	            IF "Tor2_RecepturyStacjaMycia".Receptura[#aktualnyNumerReceptury].Krok[#aktualnyKrokMycia].PM[2] = 0
	            THEN
	                ;
	                "Tor2_program".program.numerKroku := 7280;
	                "Tor2_RecepturyStacjaMycia".numerKrokuMycia :=
	                "Tor2_RecepturyStacjaMycia".numerKrokuMycia + 1;
	            END_IF;
	            
	            
	            ;
	            IF "Cip".obiekt["Cip".tor[2].przewodnośćNaPowrocie].WartośćPomiaru <=
	                "Tor2_RecepturyStacjaMycia".Receptura[#aktualnyNumerReceptury].Krok[#aktualnyKrokMycia].PM[12] +
	                "Tor2_RecepturyStacjaMycia".Receptura[#aktualnyNumerReceptury].Krok[#aktualnyKrokMycia].PM[15]
	                
	            THEN
	                "Cip".obiekt["Cip".tor[2].przepływomierzZaWymiennikiem].zerujLicznik1 := 0;
	                "Cip".obiekt["Cip".tor[2].przepływomierzZaWymiennikiem].startLicznik1 := 1;
	            ELSE
	                "Cip".obiekt["Cip".tor[2].przepływomierzZaWymiennikiem].startLicznik1 := 0;
	            END_IF;
	            
	            IF "Cip".obiekt["Cip".tor[2].przepływomierzZaWymiennikiem].licznik1 >
	                "Tor2_RecepturyStacjaMycia".Receptura[#aktualnyNumerReceptury].Krok[#aktualnyKrokMycia].PM[5]
	            THEN
	                "Cip".obiekt["Cip".tor[2].przepływomierzZaWymiennikiem].zerujLicznik1 := 0;
	                "Cip".obiekt["Cip".tor[2].przepływomierzZaWymiennikiem].startLicznik1 := 0;
	              
	                
	                "linia1_pompa_zezwolenie" := 0;
	                "IdźDoKroku"(inNumerKrokuDocelowy := 7271,
	                             inZadaneOpóżnienie := 9,
	                             numerKroku := "Tor2_program".program.numerKroku,
	                             opóźnienie := "Tor2_program".program.opóżnienie,
	                             pauza := "Tor2_hmi".button.bPauza.set);
	                
	                
	              
	            END_IF;
	            
	            
	            "Tor2_program".program.zadana1 := "Tor2_RecepturyStacjaMycia".Receptura[#aktualnyNumerReceptury].Krok[#aktualnyKrokMycia].PM[12] +
	            "Tor2_RecepturyStacjaMycia".Receptura[#aktualnyNumerReceptury].Krok[#aktualnyKrokMycia].PM[15];
	            "Tor2_program".program.aktualna1 := "Cip".obiekt["Cip".tor[2].przewodnośćNaPowrocie].WartośćPomiaru;
	            "Tor2_program".program.zadana2 := "Tor2_RecepturyStacjaMycia".Receptura[#aktualnyNumerReceptury].Krok[#aktualnyKrokMycia].PM[5];
	            "Tor2_program".program.aktualna2 := "Cip".obiekt["Cip".tor[2].przepływomierzZaWymiennikiem].licznik1;
	        7271:
	            
	            "Tor2_RecepturyStacjaMycia".numerKrokuMycia :=
	            "Tor2_RecepturyStacjaMycia".numerKrokuMycia + 1;
	            "Cip".obiekt["Cip".tor[2].przepływomierzZaWymiennikiem].licznik1 := 0;
	            "Tor2_program".program.numerKroku := 7280;
	            
	        7280://Uruchomienie dezynfekcji
	            "Tor2_RecepturyStacjaMycia".numerKrokuMycia := 6;
	            IF "Tor2_RecepturyStacjaMycia".Receptura[#aktualnyNumerReceptury].Krok[#aktualnyKrokMycia].PM[1] = 0
	                OR (#aktualnyKrokMycia = 6 AND "Tor2_hmi".bPomińDesynfekcje)
	            THEN
	                
	                
	                "IdźDoKroku"(inNumerKrokuDocelowy := 7289,
	                             inZadaneOpóżnienie := 30,
	                             numerKroku := "Tor2_program".program.numerKroku,
	                             opóźnienie := "Tor2_program".program.opóżnienie,
	                             pauza := "Tor2_hmi".button.bPauza.set);
	                
	            ELSE
	                "IdźDoKroku"(inNumerKrokuDocelowy := 7281,
	                             inZadaneOpóżnienie := 30,
	                             numerKroku := "Tor2_program".program.numerKroku,
	                             opóźnienie := "Tor2_program".program.opóżnienie,
	                             pauza := "Tor2_hmi".button.bPauza.set);
	            END_IF;
	            
	            
	        7281://napełnianie zbironika dezynfekcji
	            
	            
	            
	            IF "Cip".obiekt["Cip".tor[2].zbiornikDezynfekantu.poziomAnalogowy].WartośćPomiaru > 50
	            THEN
	                
	                
	                "IdźDoKroku"(inNumerKrokuDocelowy := 7282,
	                             inZadaneOpóżnienie := 1,
	                             numerKroku := "Tor2_program".program.numerKroku,
	                             opóźnienie := "Tor2_program".program.opóżnienie,
	                             pauza := "Tor2_hmi".button.bPauza.set);
	            END_IF;
	            "Tor2_program".program.zadana1 := 50;
	            "Tor2_program".program.aktualna1 := "Cip".obiekt["Cip".tor[2].zbiornikDezynfekantu.poziomAnalogowy].WartośćPomiaru;
	            "Tor2_program".program.zadana2 := 0;
	            "Tor2_program".program.aktualna2 := 0;
	            "Cip".obiekt["Cip".tor[2].przepływomierzZaWymiennikiem].licznik1 := 0;
	            
	        7282://dozowanie dezynfekanta
	            "IdźDoKroku"(inNumerKrokuDocelowy := 7283,
	                         inZadaneOpóżnienie := "Tor2_RecepturyStacjaMycia".Receptura[#aktualnyNumerReceptury].Krok[#aktualnyKrokMycia].PM[20],
	                         numerKroku := "Tor2_program".program.numerKroku,
	                         opóźnienie := "Tor2_program".program.opóżnienie,
	                         pauza := "Tor2_hmi".button.bPauza.set);
	            
	            //jeżeli nie leci dezynfekant to kasuj czas dozowania
	            IF "Cip".obiekt["Cip".tor[0].zbiorniczekDozowanieDezynfekantu.czujnikDolnegoPoziomu].hmiPotwWysterowania = 0 THEN
	                "Tor2_program".program.opóżnienie := "Tor2_program".program.opóżnienie - 0.1;
	            END_IF;
	            
	            "Tor2_program".program.zadana1 := "Tor2_RecepturyStacjaMycia".Receptura[#aktualnyNumerReceptury].Krok[#aktualnyKrokMycia].PM[20];
	            "Tor2_program".program.aktualna1 := "Tor2_program".program.opóżnienie;
	            "Tor2_program".program.zadana2 := 0;
	            "Tor2_program".program.aktualna2 := 0;
	            "Cip".obiekt["Cip".tor[2].przepływomierzZaWymiennikiem].licznik1 := 0;
	            
	        7283://dezynfekcja chemiczna
	            "IdźDoKroku"(inNumerKrokuDocelowy := 7284,
	                         inZadaneOpóżnienie := "Tor2_RecepturyStacjaMycia".Receptura[#aktualnyNumerReceptury].Krok[6].PM[6], //czas mycia
	                         numerKroku := "Tor2_program".program.numerKroku,
	                         opóźnienie := "Tor2_program".program.opóżnienie,
	                         pauza := "Tor2_hmi".button.bPauza.set);
	            
	            "Tor2_program".program.zadana1 := "Tor2_RecepturyStacjaMycia".Receptura[#aktualnyNumerReceptury].Krok[6].PM[6];
	            "Tor2_program".program.aktualna1 := "Tor2_program".program.opóżnienie;
	            "Tor2_program".program.zadana2 := 0;
	            "Tor2_program".program.aktualna2 := 0;
	            "Cip".obiekt["Cip".tor[2].przepływomierzZaWymiennikiem].licznik1 := 0;
	            
	        7284://oprożnianie zbiornika dezynfekcji
	            
	            IF "Cip".obiekt["Cip".tor[2].zbiornikDezynfekantu.czujnikDolnegoPoziomu].hmiPotwWysterowania = 0
	            THEN
	                
	                "IdźDoKroku"(inNumerKrokuDocelowy := 7287,
	                             inZadaneOpóżnienie := 2,
	                             numerKroku := "Tor2_program".program.numerKroku,
	                             opóźnienie := "Tor2_program".program.opóżnienie,
	                             pauza := "Tor2_hmi".button.bPauza.set);
	            END_IF;
	            "Tor2_program".program.zadana1 := 0;
	            "Tor2_program".program.aktualna1 := BOOL_TO_INT("Cip".obiekt["Cip".tor[2].zbiornikDezynfekantu.czujnikDolnegoPoziomu].hmiPotwWysterowania);
	            "Tor2_program".program.zadana2 := 0;
	            "Tor2_program".program.aktualna2 := 0;
	            "Cip".obiekt["Cip".tor[2].przepływomierzZaWymiennikiem].licznik1 := 0;
	            
	            
	            
	            
	        7287://Płukanie poo dezynfekcji   
	            
	            
	            IF "Tor2_hmi".bPomińDesynfekcje = 1
	            THEN
	                "Tor2_program".program.numerKroku := 7290;
	            END_IF;
	            
	            "Cip".obiekt["Cip".tor[2].przepływomierzZaWymiennikiem].zerujLicznik1 := 0;
	            "Cip".obiekt["Cip".tor[2].przepływomierzZaWymiennikiem].startLicznik1 := 1;
	            
	            
	            IF "Cip".obiekt["Cip".tor[2].przepływomierzZaWymiennikiem].licznik1 >
	                "Tor2_RecepturyStacjaMycia".Receptura[#aktualnyNumerReceptury].Krok[#aktualnyKrokMycia].PM[5]
	            THEN
	                "Cip".obiekt["Cip".tor[2].przepływomierzZaWymiennikiem].zerujLicznik1 := 0;
	                "Cip".obiekt["Cip".tor[2].przepływomierzZaWymiennikiem].startLicznik1 := 0;
	                "Cip".obiekt["Cip".tor[2].przepływomierzZaWymiennikiem].licznik1 := 0;
	                "Tor2_program".program.numerKroku := 7289;
	            END_IF;
	            
	            
	            
	            "Tor2_program".program.zadana1 := "Tor2_RecepturyStacjaMycia".Receptura[#aktualnyNumerReceptury].Krok[#aktualnyKrokMycia].PM[5];
	            "Tor2_program".program.aktualna1 := "Cip".obiekt["Cip".tor[2].przepływomierzZaWymiennikiem].licznik1;
	            "Tor2_program".program.zadana2 := 0;
	            "Tor2_program".program.aktualna2 := 0;
	            
	        7289://Drenaż zbiornika
	            
	            IF "Tor2_RecepturyStacjaMycia".Receptura[#aktualnyNumerReceptury].Krok[#aktualnyKrokMycia].PM[23] = 0
	            THEN
	                "Tor2_program".program.numerKroku := 7290;
	            END_IF;
	            
	            IF
	                "Cip".obiekt["Cip".tor[2].czujnikPrzepływuNaPowrocie].hmiPotwWysterowania = 1
	            THEN
	                "Tor2_program".program.opóżnienie := 0;
	            END_IF;
	            "IdźDoKroku"(inNumerKrokuDocelowy := 7290,
	                         inZadaneOpóżnienie := "Tor2_RecepturyStacjaMycia".Receptura[#aktualnyNumerReceptury].Krok[#aktualnyKrokMycia].PM[7],
	                         numerKroku := "Tor2_program".program.numerKroku,
	                         opóźnienie := "Tor2_program".program.opóżnienie,
	                         pauza := "Tor2_hmi".button.bPauza.set);
	            
	            "Tor2_program".program.zadana1 := "Tor2_RecepturyStacjaMycia".Receptura[#aktualnyNumerReceptury].Krok[#aktualnyKrokMycia].PM[7];
	            "Tor2_program".program.aktualna1 := "Tor2_program".program.opóżnienie;
	            "Tor2_program".program.zadana2 := 0;
	            "Tor2_program".program.aktualna2 := INT_TO_REAL(BOOL_TO_INT("Cip".obiekt["Cip".tor[2].czujnikPrzepływuNaPowrocie].hmiPotwWysterowania = 1)) * 1.0;
	            
	            
	            
	        7290://zatrzymanie przepływu
	            
	            IF "Cip".obiekt["Cip".tor[2].przepływomierzZaWymiennikiem].WartośćPomiaru <5.0
	            THEN
	                "IdźDoKroku"(inNumerKrokuDocelowy := 7291,
	                             inZadaneOpóżnienie   := 10,
	                             numerKroku           := "Tor2_program".program.numerKroku,
	                             opóźnienie           := "Tor2_program".program.opóżnienie,
	                             pauza:=  "Tor2_hmi".button.bPauza.set);
	            END_IF;
	            
	            "Tor2_program".program.zadana1 := "Tor2_RecepturyStacjaMycia".Receptura[#aktualnyNumerReceptury].Krok[#aktualnyKrokMycia].PM[2];
	            "Tor2_program".program.aktualna1 := "Cip".obiekt["Cip".tor[2].przepływomierzZaWymiennikiem].WartośćPomiaru;
	            "Tor2_program".program.zadana2 :=5;
	            "Tor2_program".program.aktualna2 := "Tor2_program".program.opóżnienie;
	            
	            
	        7291:// odlicz opóźnienie
	            
	            "IdźDoKroku"(inNumerKrokuDocelowy := 7100,
	                         inZadaneOpóżnienie   := 1,
	                         numerKroku           := "Tor2_program".program.numerKroku,
	                         opóźnienie           := "Tor2_program".program.opóżnienie,
	                         pauza:=  "Tor2_hmi".button.bPauza.set);
	            "Tor2_hmi".button.bStop.set := 1;
	          
	            
	            
	        "Tor2_program".program.zadana1 := 0;
	        "Tor2_program".program.aktualna1 :=0;
	        "Tor2_program".program.zadana2 := 10;
	        "Tor2_program".program.aktualna2 := "Tor2_program".program.opóżnienie;
	            
	    7300: //Zaczytanie numeru receptury - krok mycia =2
	        
	        IF "Tor2_RecepturyStacjaMycia".bPokazOknoWyboruReceptury = 0 THEN
	            "Tor2_RecepturyStacjaMycia".bPokazOknoWyboruReceptury := 1;
	        END_IF;
	        IF
	            "Tor2_RecepturyStacjaMycia".klawiszUżyjTejReceptury = 1
	            AND "Tor2_RecepturyStacjaMycia".numerWyswietlanejReceptury = 1
	        THEN
	            "IdźDoKroku"(inNumerKrokuDocelowy := 7301,
	                         inZadaneOpóżnienie   := 0,
	                         numerKroku           := "Tor2_program".program.numerKroku,
	                         opóźnienie           := "Tor2_program".program.opóżnienie,
	                         pauza:=  "Tor2_hmi".button.bPauza.set);
	            "Tor2_RecepturyStacjaMycia".bPokazOknoWyboruReceptury := 0;
	            "Tor2_RecepturyStacjaMycia".numerKrokuMycia := 3;
	            #doSkasowania := 1;
	            
	        END_IF;
	        "Tor2_program".program.zadana1 := 0;
	        "Tor2_program".program.aktualna1 := 0;
	        "Tor2_program".program.zadana2 := 0;
	        "Tor2_program".program.aktualna2 := 0;
	            
	    7301://kolejny krok mycia
	      
	        IF
	            "Tor2_RecepturyStacjaMycia".numerKrokuMycia < 5
	        THEN
	            "IdźDoKroku"(inNumerKrokuDocelowy := 7310,
	                         inZadaneOpóżnienie   := 1,
	                         numerKroku           := "Tor2_program".program.numerKroku,
	                         opóźnienie           := "Tor2_program".program.opóżnienie,
	                         pauza:=  "Tor2_hmi".button.bPauza.set);
	        END_IF;
	        IF
	            "Tor2_RecepturyStacjaMycia".numerKrokuMycia >=5
	        THEN
	            "IdźDoKroku"(inNumerKrokuDocelowy := 7290,
	                         inZadaneOpóżnienie   := 1,
	                         numerKroku           := "Tor2_program".program.numerKroku,
	                         opóźnienie           := "Tor2_program".program.opóżnienie,
	                         pauza:=  "Tor2_hmi".button.bPauza.set);
	            "Tor2_hmi".button.bCip.set := 0;
	        END_IF;
	        "Tor2_program".program.zadana1 := 0;
	        "Tor2_program".program.aktualna1 := 0;
	        "Tor2_program".program.zadana2 := 0;
	        "Tor2_program".program.aktualna2 := 0;
	        
	        
	    7310:// Uzupełnianie poziomu w zbiorniku
	        
	        IF
	            "Tor2_RecepturyStacjaMycia".numerKrokuMycia = 3
	        THEN
	            IF "Cip".obiekt["Cip".tor[0].zbiornikŁugu.czujnikDolnegoPoziomu].hmiPotwWysterowania = 1 THEN
	                "IdźDoKroku"(inNumerKrokuDocelowy := 7320,
	                             inZadaneOpóżnienie   := 1,
	                             numerKroku           := "Tor2_program".program.numerKroku,
	                             opóźnienie           := "Tor2_program".program.opóżnienie,
	                             pauza:=  "Tor2_hmi".button.bPauza.set);
	            END_IF;
	        END_IF;
	        IF
	            "Tor2_RecepturyStacjaMycia".numerKrokuMycia = 4
	        THEN
	            IF "Cip".obiekt["Cip".tor[0].zbiornikKwasu.czujnikDolnegoPoziomu].hmiPotwWysterowania = 1 THEN
	                "IdźDoKroku"(inNumerKrokuDocelowy := 7320,
	                             inZadaneOpóżnienie   := 1,
	                             numerKroku           := "Tor2_program".program.numerKroku,
	                             opóźnienie           := "Tor2_program".program.opóżnienie,
	                             pauza:=  "Tor2_hmi".button.bPauza.set);
	            END_IF;
	        END_IF;
	            
	        "Tor2_program".program.zadana1 :=1;
	        "Tor2_program".program.aktualna1 :=BOOL_TO_INT("Cip".obiekt["Cip".tor[0].zbiornikŁugu.czujnikDolnegoPoziomu].hmiPotwWysterowania);
	        "Tor2_program".program.zadana2 := 1;
	        "Tor2_program".program.aktualna2 := BOOL_TO_INT("Cip".obiekt["Cip".tor[0].zbiornikKwasu.czujnikDolnegoPoziomu].hmiPotwWysterowania);
	        
	    7320://przygotowanie środkla chemicznego
	        
	        IF "Cip".obiekt["Cip".tor[2].przewodnośćNaPowrocie].WartośćPomiaru >=
	            "Tor2_RecepturyStacjaMycia".Receptura[#aktualnyNumerReceptury].Krok[#aktualnyKrokMycia].PM[10] +
	            "Tor2_RecepturyStacjaMycia".Receptura[#aktualnyNumerReceptury].Krok[#aktualnyKrokMycia].PM[15]
	            AND
	            "Cip".obiekt["Cip".tor[2].temperaturaNaPowrocie].WartośćPomiaru >=
	            "Tor2_RecepturyStacjaMycia".Receptura[#aktualnyNumerReceptury].Krok[#aktualnyKrokMycia].PM[13] -
	            "Tor2_RecepturyStacjaMycia".Receptura[#aktualnyNumerReceptury].Krok[#aktualnyKrokMycia].PM[16]
	        THEN
	            "IdźDoKroku"(inNumerKrokuDocelowy := 7321,
	                         inZadaneOpóżnienie   := 30,
	                         numerKroku           := "Tor2_program".program.numerKroku,
	                         opóźnienie           := "Tor2_program".program.opóżnienie,
	                         pauza:=  "Tor2_hmi".button.bPauza.set);
	            
	        END_IF;
	        
	        "Tor2_program".program.zadana1 := "Tor2_RecepturyStacjaMycia".Receptura[#aktualnyNumerReceptury].Krok[#aktualnyKrokMycia].PM[10] +
	        "Tor2_RecepturyStacjaMycia".Receptura[#aktualnyNumerReceptury].Krok[#aktualnyKrokMycia].PM[15];
	        "Tor2_program".program.aktualna1 := "Cip".obiekt["Cip".tor[2].przewodnośćNaPowrocie].WartośćPomiaru;
	        "Tor2_program".program.zadana2 :=  "Tor2_RecepturyStacjaMycia".Receptura[#aktualnyNumerReceptury].Krok[#aktualnyKrokMycia].PM[13] -
	        "Tor2_RecepturyStacjaMycia".Receptura[#aktualnyNumerReceptury].Krok[#aktualnyKrokMycia].PM[16];
	        "Tor2_program".program.aktualna2 := "Cip".obiekt["Cip".tor[2].temperaturaNaPowrocie].WartośćPomiaru;
	        
	        
	        
	    7321://wypłukiwanie środka chemicznego
	        
	        IF "Cip".obiekt["Cip".tor[2].przewodnośćNaPowrocie].WartośćPomiaru <
	            "Tor2_RecepturyStacjaMycia".Receptura[#aktualnyNumerReceptury].Krok[#aktualnyKrokMycia].PM[10] -
	            "Tor2_RecepturyStacjaMycia".Receptura[#aktualnyNumerReceptury].Krok[#aktualnyKrokMycia].PM[15]
	        THEN
	            "IdźDoKroku"(inNumerKrokuDocelowy := 7330,
	                         inZadaneOpóżnienie   := 0,
	                         numerKroku           := "Tor2_program".program.numerKroku,
	                         opóźnienie           := "Tor2_program".program.opóżnienie,
	                         pauza:=  "Tor2_hmi".button.bPauza.set);
	        END_IF;
	        
	        "Tor2_program".program.zadana1 := "Tor2_RecepturyStacjaMycia".Receptura[#aktualnyNumerReceptury].Krok[#aktualnyKrokMycia].PM[10] -
	        "Tor2_RecepturyStacjaMycia".Receptura[#aktualnyNumerReceptury].Krok[#aktualnyKrokMycia].PM[15];
	        "Tor2_program".program.aktualna1 := "Cip".obiekt["Cip".tor[2].przewodnośćNaPowrocie].WartośćPomiaru;
	        "Tor2_program".program.zadana2 := "Tor2_RecepturyStacjaMycia".Receptura[#aktualnyNumerReceptury].Krok[#aktualnyKrokMycia].PM[13] -
	        "Tor2_RecepturyStacjaMycia".Receptura[#aktualnyNumerReceptury].Krok[#aktualnyKrokMycia].PM[16];
	        "Tor2_program".program.aktualna2 := "Cip".obiekt["Cip".tor[2].przewodnośćNaPowrocie].WartośćPomiaru;
	        
	        
	    7330://koniec mycia
	        
	        "IdźDoKroku"(inNumerKrokuDocelowy := 7301,
	                     inZadaneOpóżnienie   := 0,
	                     numerKroku           := "Tor2_program".program.numerKroku,
	                     opóźnienie           := "Tor2_program".program.opóżnienie,
	                     pauza:=  "Tor2_hmi".button.bPauza.set);
	        "Tor2_RecepturyStacjaMycia".numerKrokuMycia :=
	        "Tor2_RecepturyStacjaMycia".numerKrokuMycia + 1;
	        
	        "Tor2_program".program.zadana1 := 0;
	        "Tor2_program".program.aktualna1 := 0;
	        "Tor2_program".program.zadana2 := 0;
	        "Tor2_program".program.aktualna2 := 0;
	        
	    7400://   Zaczytanie numeru receptury (program ustawia Krok mycia = 1) tylko program numer 2
	        
	        IF "Tor2_RecepturyStacjaMycia".bPokazOknoWyboruReceptury = 0 THEN
	            "Tor2_RecepturyStacjaMycia".bPokazOknoWyboruReceptury := 1;
	        END_IF;
	        IF
	            "Tor2_RecepturyStacjaMycia".klawiszUżyjTejReceptury = 1
	            AND "Tor2_RecepturyStacjaMycia".numerWyswietlanejReceptury = 2
	        THEN
	            "IdźDoKroku"(inNumerKrokuDocelowy := 7401,
	                         inZadaneOpóżnienie   := 0,
	                         numerKroku           := "Tor2_program".program.numerKroku,
	                         opóźnienie           := "Tor2_program".program.opóżnienie,
	                         pauza:=  "Tor2_hmi".button.bPauza.set);
	            "Tor2_RecepturyStacjaMycia".bPokazOknoWyboruReceptury := 0;
	            "Tor2_RecepturyStacjaMycia".numerKrokuMycia := 1;
	            #doSkasowania := 1;
	            
	            //Wyskakuje okno wyboru receptur mycia (można wybrać tylko program 2),
	            //po wybraniu krok przechodzi
	            //(program blokuje możliwość pracy na drugim torze - może mrygać na nim kontrolka CIP)
	            //do zrobienia !!!!!
	            
	            
	        END_IF;
	        "Tor2_program".program.zadana1 := 0;
	        "Tor2_program".program.aktualna1 := 0;
	        "Tor2_program".program.zadana2 := 0;
	        "Tor2_program".program.aktualna2 := 0;
	        
	        
	    7401:// drenaż zbiornika wody wtórnej
	        
	        
	        IF
	            "Cip".obiekt["Cip".tor[2].czujnikPrzepływuNaPowrocie].hmiPotwWysterowania = 1
	        THEN
	            "Tor2_program".program.opóżnienie := 0;
	        END_IF;
	        "IdźDoKroku"(inNumerKrokuDocelowy := 7402,
	                     inZadaneOpóżnienie   := "Tor2_RecepturyStacjaMycia".Receptura[#aktualnyNumerReceptury].Krok[#aktualnyKrokMycia].PM[7],
	                     numerKroku           := "Tor2_program".program.numerKroku,
	                     opóźnienie           := "Tor2_program".program.opóżnienie,
	                     pauza:=  "Tor2_hmi".button.bPauza.set);
	        
	        "Tor2_program".program.zadana1 := "Tor2_RecepturyStacjaMycia".Receptura[#aktualnyNumerReceptury].Krok[#aktualnyKrokMycia].PM[7];
	        "Tor2_program".program.aktualna1 := "Tor2_program".program.opóżnienie;
	        "Tor2_program".program.zadana2 := 0;
	        "Tor2_program".program.aktualna2 := INT_TO_REAL(BOOL_TO_INT("Cip".obiekt["Cip".tor[2].czujnikPrzepływuNaPowrocie].hmiPotwWysterowania = 1)) * 1.0;
	        
	    7402://płukanie zimne
	            
	        IF "Tor2_RecepturyStacjaMycia".Receptura[#aktualnyNumerReceptury].Krok[#aktualnyKrokMycia].PM[2] = 0
	            THEN
	                ;
	                "Tor2_program".program.numerKroku := 7403;
	                "Tor2_RecepturyStacjaMycia".numerKrokuMycia :=
	                "Tor2_RecepturyStacjaMycia".numerKrokuMycia + 1;
	            END_IF;
	            
	            
	            ;
	            IF "Cip".obiekt["Cip".tor[2].przewodnośćNaPowrocie].WartośćPomiaru <=
	                "Tor2_RecepturyStacjaMycia".Receptura[#aktualnyNumerReceptury].Krok[#aktualnyKrokMycia].PM[12] +
	                "Tor2_RecepturyStacjaMycia".Receptura[#aktualnyNumerReceptury].Krok[#aktualnyKrokMycia].PM[14]
	            THEN
	                "Cip".obiekt["Cip".tor[2].przepływomierzZaWymiennikiem].zerujLicznik1 := 0;
	                "Cip".obiekt["Cip".tor[2].przepływomierzZaWymiennikiem].startLicznik1 := 1;
	            ELSE
	                "Cip".obiekt["Cip".tor[2].przepływomierzZaWymiennikiem].startLicznik1 := 0;
	            END_IF;
	            
	            IF "Cip".obiekt["Cip".tor[2].przepływomierzZaWymiennikiem].licznik1 >
	                "Tor2_RecepturyStacjaMycia".Receptura[#aktualnyNumerReceptury].Krok[#aktualnyKrokMycia].PM[5]
	            THEN
	                "Cip".obiekt["Cip".tor[2].przepływomierzZaWymiennikiem].zerujLicznik1 := 0;
	                "Cip".obiekt["Cip".tor[2].przepływomierzZaWymiennikiem].startLicznik1 := 0;
	                "Cip".obiekt["Cip".tor[2].przepływomierzZaWymiennikiem].licznik1 := 0;
	                "Tor2_program".program.numerKroku := 7403;
	                "Tor2_RecepturyStacjaMycia".numerKrokuMycia :=
	                "Tor2_RecepturyStacjaMycia".numerKrokuMycia + 1;
	            END_IF;
	            
	            
	            "Tor2_program".program.zadana1 := "Tor2_RecepturyStacjaMycia".Receptura[#aktualnyNumerReceptury].Krok[#aktualnyKrokMycia].PM[12] +
	            "Tor2_RecepturyStacjaMycia".Receptura[#aktualnyNumerReceptury].Krok[#aktualnyKrokMycia].PM[14];
	            "Tor2_program".program.aktualna1 := "Cip".obiekt["Cip".tor[2].przewodnośćNaPowrocie].WartośćPomiaru;
	            "Tor2_program".program.zadana2 := "Tor2_RecepturyStacjaMycia".Receptura[#aktualnyNumerReceptury].Krok[#aktualnyKrokMycia].PM[5];
	            "Tor2_program".program.aktualna2 := "Cip".obiekt["Cip".tor[2].przepływomierzZaWymiennikiem].licznik1;
	            
	        7403: //płukanie ciepłe
	            
	            IF "Tor2_RecepturyStacjaMycia".Receptura[#aktualnyNumerReceptury].Krok[#aktualnyKrokMycia].PM[2] = 0
	            THEN
	                ;
	                "Tor2_program".program.numerKroku := 7404;
	                "Tor2_RecepturyStacjaMycia".numerKrokuMycia :=
	                "Tor2_RecepturyStacjaMycia".numerKrokuMycia + 1;
	            END_IF;
	            
	            
	            ;
	            IF "Cip".obiekt["Cip".tor[2].przewodnośćNaPowrocie].WartośćPomiaru <=
	                "Tor2_RecepturyStacjaMycia".Receptura[#aktualnyNumerReceptury].Krok[#aktualnyKrokMycia].PM[12] +
	                "Tor2_RecepturyStacjaMycia".Receptura[#aktualnyNumerReceptury].Krok[#aktualnyKrokMycia].PM[15]
	                AND
	                "Cip".obiekt["Cip".tor[2].temperaturaNaPowrocie].WartośćPomiaru >=
	                "Tor2_RecepturyStacjaMycia".Receptura[#aktualnyNumerReceptury].Krok[#aktualnyKrokMycia].PM[14] -
	                "Tor2_RecepturyStacjaMycia".Receptura[#aktualnyNumerReceptury].Krok[#aktualnyKrokMycia].PM[16]
	                
	            THEN
	                "Cip".obiekt["Cip".tor[2].przepływomierzZaWymiennikiem].zerujLicznik1 := 0;
	                "Cip".obiekt["Cip".tor[2].przepływomierzZaWymiennikiem].startLicznik1 := 1;
	            ELSE
	                "Cip".obiekt["Cip".tor[2].przepływomierzZaWymiennikiem].startLicznik1 := 0;
	            END_IF;
	            
	            IF "Cip".obiekt["Cip".tor[2].przepływomierzZaWymiennikiem].licznik1 >
	                "Tor2_RecepturyStacjaMycia".Receptura[#aktualnyNumerReceptury].Krok[#aktualnyKrokMycia].PM[5]
	            THEN
	                "Cip".obiekt["Cip".tor[2].przepływomierzZaWymiennikiem].zerujLicznik1 := 0;
	                "Cip".obiekt["Cip".tor[2].przepływomierzZaWymiennikiem].startLicznik1 := 0;
	                "Cip".obiekt["Cip".tor[2].przepływomierzZaWymiennikiem].licznik1 := 0;
	                "Tor2_program".program.numerKroku := 7404;
	                "Tor2_RecepturyStacjaMycia".numerKrokuMycia :=
	                "Tor2_RecepturyStacjaMycia".numerKrokuMycia + 1;
	            END_IF;
	            
	            
	            "Tor2_program".program.zadana1 := "Tor2_RecepturyStacjaMycia".Receptura[#aktualnyNumerReceptury].Krok[#aktualnyKrokMycia].PM[14] -
	            "Tor2_RecepturyStacjaMycia".Receptura[#aktualnyNumerReceptury].Krok[#aktualnyKrokMycia].PM[16];
	            "Tor2_program".program.aktualna1 := "Cip".obiekt["Cip".tor[2].temperaturaNaPowrocie].WartośćPomiaru;
	            "Tor2_program".program.zadana2 := "Tor2_RecepturyStacjaMycia".Receptura[#aktualnyNumerReceptury].Krok[#aktualnyKrokMycia].PM[5];
	            "Tor2_program".program.aktualna2 := "Cip".obiekt["Cip".tor[2].przepływomierzZaWymiennikiem].licznik1;
	            
	        7404://drenaż zbiornika
	            
	            IF
	                "Cip".obiekt["Cip".tor[2].czujnikPrzepływuNaPowrocie].hmiPotwWysterowania = 1
	            THEN
	                "Tor2_program".program.opóżnienie := 0;
	            END_IF;
	            "IdźDoKroku"(inNumerKrokuDocelowy := 7405,
	                         inZadaneOpóżnienie   := "Tor2_RecepturyStacjaMycia".Receptura[#aktualnyNumerReceptury].Krok[#aktualnyKrokMycia].PM[7],
	                         numerKroku           := "Tor2_program".program.numerKroku,
	                         opóźnienie           := "Tor2_program".program.opóżnienie,
	                         pauza:=  "Tor2_hmi".button.bPauza.set);
	            IF "Tor2_program".program.opóżnienie
	                >= "Tor2_RecepturyStacjaMycia".Receptura[#aktualnyNumerReceptury].Krok[#aktualnyKrokMycia].PM[7]
	            THEN
	                "Tor2_RecepturyStacjaMycia".numerKrokuMycia :=
	                "Tor2_RecepturyStacjaMycia".numerKrokuMycia + 1;
	            END_IF;
	            "Tor2_program".program.zadana1 := "Tor2_RecepturyStacjaMycia".Receptura[#aktualnyNumerReceptury].Krok[#aktualnyKrokMycia].PM[7];
	            "Tor2_program".program.aktualna1 := "Tor2_program".program.opóżnienie;
	            "Tor2_program".program.zadana2 := 0;
	            "Tor2_program".program.aktualna2 := INT_TO_REAL(BOOL_TO_INT("Cip".obiekt["Cip".tor[2].czujnikPrzepływuNaPowrocie].hmiPotwWysterowania = 1)) * 1.0;
	        
	        7405:// zaczytanie kroku
	      
	            
	            
	            IF "Tor2_RecepturyStacjaMycia".numerKrokuMycia>=5
	            THEN
	                ;
	                "Tor2_program".program.numerKroku := 7420;
	            ELSE
	                "IdźDoKroku"(inNumerKrokuDocelowy := 7410,
	                             inZadaneOpóżnienie   :=0,
	                             numerKroku           := "Tor2_program".program.numerKroku,
	                             opóźnienie           := "Tor2_program".program.opóżnienie,
	                             pauza:=  "Tor2_hmi".button.bPauza.set);
	            END_IF;
	            
	        7410://drenaż zbiornika
	            
	                
	            IF "Tor2_RecepturyStacjaMycia".Receptura[#aktualnyNumerReceptury].Krok[#aktualnyKrokMycia].PM[2] = 0
	                THEN
	                    ;
	                    "Tor2_program".program.numerKroku := 7415;
	               
	                END_IF;
	            
	            IF
	                "Cip".obiekt["Cip".tor[2].czujnikPrzepływuNaPowrocie].hmiPotwWysterowania = 1
	            THEN
	                "Tor2_program".program.opóżnienie := 0;
	            END_IF;
	            "IdźDoKroku"(inNumerKrokuDocelowy := 7411,
	                         inZadaneOpóżnienie   := "Tor2_RecepturyStacjaMycia".Receptura[#aktualnyNumerReceptury].Krok[#aktualnyKrokMycia].PM[7],
	                         numerKroku           := "Tor2_program".program.numerKroku,
	                         opóźnienie           := "Tor2_program".program.opóżnienie,
	                         pauza:=  "Tor2_hmi".button.bPauza.set);
	            
	            "Tor2_program".program.zadana1 := "Tor2_RecepturyStacjaMycia".Receptura[#aktualnyNumerReceptury].Krok[#aktualnyKrokMycia].PM[7];
	            "Tor2_program".program.aktualna1 := "Tor2_program".program.opóżnienie;
	            "Tor2_program".program.zadana2 := 0;
	            "Tor2_program".program.aktualna2 := INT_TO_REAL(BOOL_TO_INT("Cip".obiekt["Cip".tor[2].czujnikPrzepływuNaPowrocie].hmiPotwWysterowania = 1)) * 1.0;
	            
	        7411: //Wypełnienie obiegu środkiem myjącym
	            
	            IF "Cip".obiekt["Cip".tor[2].przewodnośćNaPowrocie].WartośćPomiaru >=
	                "Tor2_RecepturyStacjaMycia".Receptura[#aktualnyNumerReceptury].Krok[#aktualnyKrokMycia].PM[10] -
	                "Tor2_RecepturyStacjaMycia".Receptura[#aktualnyNumerReceptury].Krok[#aktualnyKrokMycia].PM[15]
	            THEN
	                "Tor2_program".program.numerKroku := 7412;
	                
	            END_IF;
	            
	            "Tor2_program".program.zadana1 := "Tor2_RecepturyStacjaMycia".Receptura[#aktualnyNumerReceptury].Krok[#aktualnyKrokMycia].PM[10] -
	            "Tor2_RecepturyStacjaMycia".Receptura[#aktualnyNumerReceptury].Krok[#aktualnyKrokMycia].PM[15];
	            "Tor2_program".program.aktualna1 := "Cip".obiekt["Cip".tor[2].przewodnośćNaPowrocie].WartośćPomiaru;
	            "Tor2_program".program.zadana2 := 0;
	            "Tor2_program".program.aktualna2 := 0;
	            
	        7412://    Odliczanie czasu mycia
	            
	            
	                
	                IF
	                    "Cip".obiekt["Cip".tor[2].przewodnośćNaPowrocie].WartośćPomiaru >=
	                    "Tor2_RecepturyStacjaMycia".Receptura[#aktualnyNumerReceptury].Krok[#aktualnyKrokMycia].PM[10] -
	                    "Tor2_RecepturyStacjaMycia".Receptura[#aktualnyNumerReceptury].Krok[#aktualnyKrokMycia].PM[15]
	                    AND
	                    "Cip".obiekt["Cip".tor[2].temperaturaNaPowrocie].WartośćPomiaru >=
	                    "Tor2_RecepturyStacjaMycia".Receptura[#aktualnyNumerReceptury].Krok[#aktualnyKrokMycia].PM[13] -
	                    "Tor2_RecepturyStacjaMycia".Receptura[#aktualnyNumerReceptury].Krok[#aktualnyKrokMycia].PM[16]
	                THEN
	                    ;
	                ELSE
	                    "Tor2_program".program.opóżnienie := "Tor2_program".program.opóżnienie -0.1;
	                END_IF;
	                "IdźDoKroku"(inNumerKrokuDocelowy := 7413,
	                             inZadaneOpóżnienie := "Tor2_RecepturyStacjaMycia".Receptura[#aktualnyNumerReceptury].Krok[#aktualnyKrokMycia].PM[6],
	                             numerKroku := "Tor2_program".program.numerKroku,
	                             opóźnienie := "Tor2_program".program.opóżnienie,
	                             pauza:=  "Tor2_hmi".button.bPauza.set);
	                
	                
	                
	                "Tor2_program".program.zadana1 := "Tor2_RecepturyStacjaMycia".Receptura[#aktualnyNumerReceptury].Krok[#aktualnyKrokMycia].PM[13] -
	                "Tor2_RecepturyStacjaMycia".Receptura[#aktualnyNumerReceptury].Krok[#aktualnyKrokMycia].PM[16];
	                "Tor2_program".program.aktualna1 := "Cip".obiekt["Cip".tor[2].temperaturaNaPowrocie].WartośćPomiaru;
	                "Tor2_program".program.zadana2 := "Tor2_RecepturyStacjaMycia".Receptura[#aktualnyNumerReceptury].Krok[#aktualnyKrokMycia].PM[6];
	                "Tor2_program".program.aktualna2 := "Tor2_program".program.opóżnienie;
	            
	            
	        7413: //Drenaż zbiornika
	        
	            IF
	                "Cip".obiekt["Cip".tor[2].czujnikPrzepływuNaPowrocie].hmiPotwWysterowania = 1
	            THEN
	                "Tor2_program".program.opóżnienie := 0;
	            END_IF;
	            "IdźDoKroku"(inNumerKrokuDocelowy := 7414,
	                         inZadaneOpóżnienie   := "Tor2_RecepturyStacjaMycia".Receptura[#aktualnyNumerReceptury].Krok[#aktualnyKrokMycia].PM[7],
	                         numerKroku           := "Tor2_program".program.numerKroku,
	                         opóźnienie           := "Tor2_program".program.opóżnienie,
	                         pauza:=  "Tor2_hmi".button.bPauza.set);
	            
	            "Tor2_program".program.zadana1 := "Tor2_RecepturyStacjaMycia".Receptura[#aktualnyNumerReceptury].Krok[#aktualnyKrokMycia].PM[7];
	            "Tor2_program".program.aktualna1 := "Tor2_program".program.opóżnienie;
	            "Tor2_program".program.zadana2 := 0;
	            "Tor2_program".program.aktualna2 := INT_TO_REAL(BOOL_TO_INT("Cip".obiekt["Cip".tor[2].czujnikPrzepływuNaPowrocie].hmiPotwWysterowania = 1)) * 1.0;
	            
	            
	            
	        7414://    Płukanie międzyfazowe
	            
	            IF
	                "Cip".obiekt["Cip".tor[2].przewodnośćNaPowrocie].WartośćPomiaru <
	                "Tor2_RecepturyStacjaMycia".Receptura[#aktualnyNumerReceptury].Krok[#aktualnyKrokMycia].PM[12] +
	                "Tor2_RecepturyStacjaMycia".Receptura[#aktualnyNumerReceptury].Krok[#aktualnyKrokMycia].PM[15]
	                AND
	                "Cip".obiekt["Cip".tor[2].temperaturaNaPowrocie].WartośćPomiaru >=
	                "Tor2_RecepturyStacjaMycia".Receptura[#aktualnyNumerReceptury].Krok[#aktualnyKrokMycia].PM[14] -
	                "Tor2_RecepturyStacjaMycia".Receptura[#aktualnyNumerReceptury].Krok[#aktualnyKrokMycia].PM[16]
	            THEN
	                "Cip".obiekt["Cip".tor[2].przepływomierzZaWymiennikiem].zerujLicznik1 := 0;
	                "Cip".obiekt["Cip".tor[2].przepływomierzZaWymiennikiem].startLicznik1 := 1;
	            ELSE
	                "Cip".obiekt["Cip".tor[2].przepływomierzZaWymiennikiem].startLicznik1 := 0;
	            END_IF;
	            
	            
	            IF "Cip".obiekt["Cip".tor[2].przepływomierzZaWymiennikiem].licznik1 >
	                "Tor2_RecepturyStacjaMycia".Receptura[#aktualnyNumerReceptury].Krok[#aktualnyKrokMycia].PM[5]
	            THEN
	                "Cip".obiekt["Cip".tor[2].przepływomierzZaWymiennikiem].zerujLicznik1 := 0;
	                "Cip".obiekt["Cip".tor[2].przepływomierzZaWymiennikiem].startLicznik1 := 0;
	                "Cip".obiekt["Cip".tor[2].przepływomierzZaWymiennikiem].licznik1 := 0;
	                "Tor2_program".program.numerKroku := 7415;
	            END_IF;
	            
	            "Tor2_program".program.zadana1 := "Tor2_RecepturyStacjaMycia".Receptura[#aktualnyNumerReceptury].Krok[#aktualnyKrokMycia].PM[14] -
	            "Tor2_RecepturyStacjaMycia".Receptura[#aktualnyNumerReceptury].Krok[#aktualnyKrokMycia].PM[16];
	            "Tor2_program".program.aktualna1 := "Cip".obiekt["Cip".tor[2].temperaturaNaPowrocie].WartośćPomiaru;
	            "Tor2_program".program.zadana2 := "Tor2_RecepturyStacjaMycia".Receptura[#aktualnyNumerReceptury].Krok[#aktualnyKrokMycia].PM[5];
	            "Tor2_program".program.aktualna2 := "Cip".obiekt["Cip".tor[2].przepływomierzZaWymiennikiem].licznik1;
	            
	            
	        7415://koniec mycia
	            
	            "IdźDoKroku"(inNumerKrokuDocelowy := 7405,
	                         inZadaneOpóżnienie   := 0,
	                         numerKroku           := "Tor2_program".program.numerKroku,
	                         opóźnienie           := "Tor2_program".program.opóżnienie,
	                         pauza:=  "Tor2_hmi".button.bPauza.set);
	            "Tor2_RecepturyStacjaMycia".numerKrokuMycia :=
	            "Tor2_RecepturyStacjaMycia".numerKrokuMycia + 1;
	            
	            "Tor2_program".program.zadana1 := 0;
	            "Tor2_program".program.aktualna1 := 0;
	            "Tor2_program".program.zadana2 := 10;
	            "Tor2_program".program.aktualna2 := "Tor2_program".program.opóżnienie;
	            
	            
	        7420:       //Płukanie główne
	            
	            IF "Tor2_RecepturyStacjaMycia".Receptura[#aktualnyNumerReceptury].Krok[#aktualnyKrokMycia].PM[2] = 0
	            THEN
	                ;
	                "Tor2_program".program.numerKroku := 7430;
	                "Tor2_RecepturyStacjaMycia".numerKrokuMycia :=1;
	            END_IF;
	            
	            
	            ;
	            IF "Cip".obiekt["Cip".tor[2].przewodnośćNaPowrocie].WartośćPomiaru <=
	                "Tor2_RecepturyStacjaMycia".Receptura[#aktualnyNumerReceptury].Krok[#aktualnyKrokMycia].PM[12] +
	                "Tor2_RecepturyStacjaMycia".Receptura[#aktualnyNumerReceptury].Krok[#aktualnyKrokMycia].PM[15]
	                
	            THEN
	                "Cip".obiekt["Cip".tor[2].przepływomierzZaWymiennikiem].zerujLicznik1 := 0;
	                "Cip".obiekt["Cip".tor[2].przepływomierzZaWymiennikiem].startLicznik1 := 1;
	            ELSE
	                "Cip".obiekt["Cip".tor[2].przepływomierzZaWymiennikiem].startLicznik1 := 0;
	            END_IF;
	            
	            IF "Cip".obiekt["Cip".tor[2].przepływomierzZaWymiennikiem].licznik1 >
	                "Tor2_RecepturyStacjaMycia".Receptura[#aktualnyNumerReceptury].Krok[#aktualnyKrokMycia].PM[5]
	            THEN
	                "Cip".obiekt["Cip".tor[2].przepływomierzZaWymiennikiem].zerujLicznik1 := 0;
	                "Cip".obiekt["Cip".tor[2].przepływomierzZaWymiennikiem].startLicznik1 := 0;
	                "Cip".obiekt["Cip".tor[2].przepływomierzZaWymiennikiem].licznik1 := 0;
	                "Tor2_program".program.numerKroku := 7430;
	                "Tor2_RecepturyStacjaMycia".numerKrokuMycia :=1;
	            END_IF;
	            
	            
	            "Tor2_program".program.zadana1 := "Tor2_RecepturyStacjaMycia".Receptura[#aktualnyNumerReceptury].Krok[#aktualnyKrokMycia].PM[12]+
	            "Tor2_RecepturyStacjaMycia".Receptura[#aktualnyNumerReceptury].Krok[#aktualnyKrokMycia].PM[15];
	            "Tor2_program".program.aktualna1 := "Cip".obiekt["Cip".tor[2].przewodnośćNaPowrocie].WartośćPomiaru;
	            "Tor2_program".program.zadana2 := "Tor2_RecepturyStacjaMycia".Receptura[#aktualnyNumerReceptury].Krok[#aktualnyKrokMycia].PM[5];
	            "Tor2_program".program.aktualna2 := "Cip".obiekt["Cip".tor[2].przepływomierzZaWymiennikiem].licznik1;
	            
	        7430://Drenaż zbiornika ługu (program ustawia K.M = 1)
	            
	            
	            "Tor2_RecepturyStacjaMycia".numerKrokuMycia := 1;
	            
	            IF
	                "Cip".obiekt["Cip".tor[2].czujnikPrzepływuNaPowrocie].hmiPotwWysterowania = 1
	            THEN
	                "Tor2_program".program.opóżnienie := 0;
	            END_IF;
	            "IdźDoKroku"(inNumerKrokuDocelowy := 7431,
	                         inZadaneOpóżnienie   := "Tor2_RecepturyStacjaMycia".Receptura[#aktualnyNumerReceptury].Krok[#aktualnyKrokMycia].PM[7],
	                         numerKroku           := "Tor2_program".program.numerKroku,
	                         opóźnienie           := "Tor2_program".program.opóżnienie,
	                         pauza:=  "Tor2_hmi".button.bPauza.set);
	            
	            "Tor2_program".program.zadana1 := "Tor2_RecepturyStacjaMycia".Receptura[#aktualnyNumerReceptury].Krok[#aktualnyKrokMycia].PM[7];
	            "Tor2_program".program.aktualna1 := "Tor2_program".program.opóżnienie;
	            "Tor2_program".program.zadana2 := 0;
	            "Tor2_program".program.aktualna2 := INT_TO_REAL(BOOL_TO_INT("Cip".obiekt["Cip".tor[2].czujnikPrzepływuNaPowrocie].hmiPotwWysterowania = 1)) * 1.0;
	            
	        7431://płukanie zimne
	            
	            
	            IF "Tor2_RecepturyStacjaMycia".Receptura[#aktualnyNumerReceptury].Krok[#aktualnyKrokMycia].PM[2] = 0
	            THEN
	                ;
	                "Tor2_program".program.numerKroku := 7432;
	                "Tor2_RecepturyStacjaMycia".numerKrokuMycia :=
	                "Tor2_RecepturyStacjaMycia".numerKrokuMycia + 1;
	            END_IF;
	            
	            
	            ;
	            IF "Cip".obiekt["Cip".tor[2].przewodnośćNaPowrocie].WartośćPomiaru <=
	                "Tor2_RecepturyStacjaMycia".Receptura[#aktualnyNumerReceptury].Krok[#aktualnyKrokMycia].PM[12] +
	                "Tor2_RecepturyStacjaMycia".Receptura[#aktualnyNumerReceptury].Krok[#aktualnyKrokMycia].PM[15]
	                
	            THEN
	                "Cip".obiekt["Cip".tor[2].przepływomierzZaWymiennikiem].zerujLicznik1 := 0;
	                "Cip".obiekt["Cip".tor[2].przepływomierzZaWymiennikiem].startLicznik1 := 1;
	            ELSE
	                "Cip".obiekt["Cip".tor[2].przepływomierzZaWymiennikiem].startLicznik1 := 0;
	            END_IF;
	            
	            IF "Cip".obiekt["Cip".tor[2].przepływomierzZaWymiennikiem].licznik1 >
	                "Tor2_RecepturyStacjaMycia".Receptura[#aktualnyNumerReceptury].Krok[#aktualnyKrokMycia].PM[5]
	            THEN
	                "Cip".obiekt["Cip".tor[2].przepływomierzZaWymiennikiem].zerujLicznik1 := 0;
	                "Cip".obiekt["Cip".tor[2].przepływomierzZaWymiennikiem].startLicznik1 := 0;
	                "Cip".obiekt["Cip".tor[2].przepływomierzZaWymiennikiem].licznik1 := 0;
	                "Tor2_program".program.numerKroku := 7432;
	                "Tor2_RecepturyStacjaMycia".numerKrokuMycia :=
	                "Tor2_RecepturyStacjaMycia".numerKrokuMycia + 1;
	            END_IF;
	            
	            
	            "Tor2_program".program.zadana1 := "Tor2_RecepturyStacjaMycia".Receptura[#aktualnyNumerReceptury].Krok[#aktualnyKrokMycia].PM[12] +
	            "Tor2_RecepturyStacjaMycia".Receptura[#aktualnyNumerReceptury].Krok[#aktualnyKrokMycia].PM[15];
	            "Tor2_program".program.aktualna1 := "Cip".obiekt["Cip".tor[2].przewodnośćNaPowrocie].WartośćPomiaru;
	            "Tor2_program".program.zadana2 := "Tor2_RecepturyStacjaMycia".Receptura[#aktualnyNumerReceptury].Krok[#aktualnyKrokMycia].PM[5];
	            "Tor2_program".program.aktualna2 := "Cip".obiekt["Cip".tor[2].przepływomierzZaWymiennikiem].licznik1;
	            
	            
	        7432://płukanie ciepłe +km
	            
	                
	            IF "Tor2_RecepturyStacjaMycia".Receptura[#aktualnyNumerReceptury].Krok[#aktualnyKrokMycia].PM[2] = 0
	                THEN
	                    ;
	                    "Tor2_program".program.numerKroku := 7433;
	                    "Tor2_RecepturyStacjaMycia".numerKrokuMycia :=4;
	                END_IF;
	                
	                
	                ;
	                IF "Cip".obiekt["Cip".tor[2].przewodnośćNaPowrocie].WartośćPomiaru <=
	                    "Tor2_RecepturyStacjaMycia".Receptura[#aktualnyNumerReceptury].Krok[#aktualnyKrokMycia].PM[12] +
	                    "Tor2_RecepturyStacjaMycia".Receptura[#aktualnyNumerReceptury].Krok[#aktualnyKrokMycia].PM[15]
	                    AND
	                    "Cip".obiekt["Cip".tor[2].temperaturaNaPowrocie].WartośćPomiaru >=
	                    "Tor2_RecepturyStacjaMycia".Receptura[#aktualnyNumerReceptury].Krok[#aktualnyKrokMycia].PM[14] -
	                    "Tor2_RecepturyStacjaMycia".Receptura[#aktualnyNumerReceptury].Krok[#aktualnyKrokMycia].PM[16]
	                THEN
	                    "Cip".obiekt["Cip".tor[2].przepływomierzZaWymiennikiem].zerujLicznik1 := 0;
	                    "Cip".obiekt["Cip".tor[2].przepływomierzZaWymiennikiem].startLicznik1 := 1;
	                ELSE
	                    "Cip".obiekt["Cip".tor[2].przepływomierzZaWymiennikiem].startLicznik1 := 0;
	                END_IF;
	                
	                IF "Cip".obiekt["Cip".tor[2].przepływomierzZaWymiennikiem].licznik1 >
	                    "Tor2_RecepturyStacjaMycia".Receptura[#aktualnyNumerReceptury].Krok[#aktualnyKrokMycia].PM[5]
	                THEN
	                    "Cip".obiekt["Cip".tor[2].przepływomierzZaWymiennikiem].zerujLicznik1 := 0;
	                    "Cip".obiekt["Cip".tor[2].przepływomierzZaWymiennikiem].startLicznik1 := 0;
	                    "Cip".obiekt["Cip".tor[2].przepływomierzZaWymiennikiem].licznik1 := 0;
	                    "Tor2_program".program.numerKroku := 7433;
	                    "Tor2_RecepturyStacjaMycia".numerKrokuMycia := 4;
	                END_IF;
	                
	                
	                "Tor2_program".program.zadana1 := "Tor2_RecepturyStacjaMycia".Receptura[#aktualnyNumerReceptury].Krok[#aktualnyKrokMycia].PM[14] -
	                "Tor2_RecepturyStacjaMycia".Receptura[#aktualnyNumerReceptury].Krok[#aktualnyKrokMycia].PM[16];
	                "Tor2_program".program.aktualna1 := "Cip".obiekt["Cip".tor[2].temperaturaNaPowrocie].WartośćPomiaru;
	                "Tor2_program".program.zadana2 := "Tor2_RecepturyStacjaMycia".Receptura[#aktualnyNumerReceptury].Krok[#aktualnyKrokMycia].PM[5];
	                "Tor2_program".program.aktualna2 := "Cip".obiekt["Cip".tor[2].przepływomierzZaWymiennikiem].licznik1;
	                
	                
	            7433://wypelnienie obiegu srodkiem myjacym
	                
	                IF "Tor2_RecepturyStacjaMycia".Receptura[#aktualnyNumerReceptury].Krok[#aktualnyKrokMycia].PM[2] = 0
	                THEN
	                    ;
	                    "Tor2_program".program.numerKroku := 7436;
	                END_IF;
	                IF
	                    "Cip".obiekt["Cip".tor[2].czujnikPrzepływuNaPowrocie].hmiPotwWysterowania = 1
	                THEN
	                    "Tor2_program".program.opóżnienie := 0;
	                END_IF;
	                "IdźDoKroku"(inNumerKrokuDocelowy := 7434,
	                             inZadaneOpóżnienie   := "Tor2_RecepturyStacjaMycia".Receptura[#aktualnyNumerReceptury].Krok[#aktualnyKrokMycia].PM[7],
	                             numerKroku           := "Tor2_program".program.numerKroku,
	                             opóźnienie           := "Tor2_program".program.opóżnienie,
	                             pauza:=  "Tor2_hmi".button.bPauza.set);
	                
	                "Tor2_program".program.zadana1 := "Tor2_RecepturyStacjaMycia".Receptura[#aktualnyNumerReceptury].Krok[#aktualnyKrokMycia].PM[7];
	                "Tor2_program".program.aktualna1 := "Tor2_program".program.opóżnienie;
	                "Tor2_program".program.zadana2 := 0;
	                "Tor2_program".program.aktualna2 := INT_TO_REAL(BOOL_TO_INT("Cip".obiekt["Cip".tor[2].czujnikPrzepływuNaPowrocie].hmiPotwWysterowania = 1)) * 1.0;
	            
	            7434://wypełnienie obiegu srodkiem myjacym kwasnym
	                
	                ;
	                IF "Cip".obiekt["Cip".tor[2].przewodnośćNaPowrocie].WartośćPomiaru >=
	                    "Tor2_RecepturyStacjaMycia".Receptura[#aktualnyNumerReceptury].Krok[#aktualnyKrokMycia].PM[10] -
	                    "Tor2_RecepturyStacjaMycia".Receptura[#aktualnyNumerReceptury].Krok[#aktualnyKrokMycia].PM[15]
	              
	                THEN
	                    "Tor2_program".program.numerKroku := 7435;
	                END_IF;
	            
	            
	            7435://Odliczanie czasu mycia
	                
	                
	                IF
	                    "Cip".obiekt["Cip".tor[2].przewodnośćNaPowrocie].WartośćPomiaru >=
	                    "Tor2_RecepturyStacjaMycia".Receptura[#aktualnyNumerReceptury].Krok[#aktualnyKrokMycia].PM[10] -
	                    "Tor2_RecepturyStacjaMycia".Receptura[#aktualnyNumerReceptury].Krok[#aktualnyKrokMycia].PM[15]
	                    AND
	                    "Cip".obiekt["Cip".tor[2].temperaturaNaPowrocie].WartośćPomiaru >=
	                    "Tor2_RecepturyStacjaMycia".Receptura[#aktualnyNumerReceptury].Krok[#aktualnyKrokMycia].PM[13] -
	                    "Tor2_RecepturyStacjaMycia".Receptura[#aktualnyNumerReceptury].Krok[#aktualnyKrokMycia].PM[16]
	                THEN
	                    ;
	                ELSE
	                    "Tor2_program".program.opóżnienie := "Tor2_program".program.opóżnienie -0.1;
	                END_IF;
	                "IdźDoKroku"(inNumerKrokuDocelowy := 7436,
	                             inZadaneOpóżnienie := "Tor2_RecepturyStacjaMycia".Receptura[#aktualnyNumerReceptury].Krok[#aktualnyKrokMycia].PM[6],
	                             numerKroku := "Tor2_program".program.numerKroku,
	                             opóźnienie := "Tor2_program".program.opóżnienie,
	                             pauza:=  "Tor2_hmi".button.bPauza.set);
	               
	                
	                
	                "Tor2_program".program.zadana1 := "Tor2_RecepturyStacjaMycia".Receptura[#aktualnyNumerReceptury].Krok[#aktualnyKrokMycia].PM[13] -
	                "Tor2_RecepturyStacjaMycia".Receptura[#aktualnyNumerReceptury].Krok[#aktualnyKrokMycia].PM[16];
	                "Tor2_program".program.aktualna1 := "Cip".obiekt["Cip".tor[2].temperaturaNaPowrocie].WartośćPomiaru;
	                "Tor2_program".program.zadana2 := "Tor2_RecepturyStacjaMycia".Receptura[#aktualnyNumerReceptury].Krok[#aktualnyKrokMycia].PM[6];
	                "Tor2_program".program.aktualna2 := "Tor2_program".program.opóżnienie;
	                
	            7436://Drenaż zbiornika (+ K.M)
	                IF
	                    "Cip".obiekt["Cip".tor[2].czujnikPrzepływuNaPowrocie].hmiPotwWysterowania = 1
	                THEN
	                    "Tor2_program".program.opóżnienie := 0;
	                END_IF;
	                "IdźDoKroku"(inNumerKrokuDocelowy := 7439,
	                             inZadaneOpóżnienie   := "Tor2_RecepturyStacjaMycia".Receptura[#aktualnyNumerReceptury].Krok[#aktualnyKrokMycia].PM[7],
	                             numerKroku           := "Tor2_program".program.numerKroku,
	                             opóźnienie           := "Tor2_program".program.opóżnienie,
	                             pauza:=  "Tor2_hmi".button.bPauza.set);
	                
	                "Tor2_program".program.zadana1 := "Tor2_RecepturyStacjaMycia".Receptura[#aktualnyNumerReceptury].Krok[#aktualnyKrokMycia].PM[7];
	                "Tor2_program".program.aktualna1 := "Tor2_program".program.opóżnienie;
	                "Tor2_program".program.zadana2 := 0;
	                "Tor2_program".program.aktualna2 := INT_TO_REAL(BOOL_TO_INT("Cip".obiekt["Cip".tor[2].czujnikPrzepływuNaPowrocie].hmiPotwWysterowania = 1)) * 1.0;
	                
	            7439:
	                "Tor2_RecepturyStacjaMycia".numerKrokuMycia := "Tor2_RecepturyStacjaMycia".numerKrokuMycia + 1;
	                "Tor2_program".program.numerKroku := 7440;
	                
	        7440://        Płukanie główne zbiornika ługu
	            
	            IF "Tor2_RecepturyStacjaMycia".Receptura[#aktualnyNumerReceptury].Krok[#aktualnyKrokMycia].PM[2] = 0
	            THEN
	                ;
	                "Tor2_program".program.numerKroku := 7450;
	            END_IF;
	            
	            
	            ;
	            IF "Cip".obiekt["Cip".tor[2].przewodnośćNaPowrocie].WartośćPomiaru <=
	                "Tor2_RecepturyStacjaMycia".Receptura[#aktualnyNumerReceptury].Krok[#aktualnyKrokMycia].PM[12] +
	                "Tor2_RecepturyStacjaMycia".Receptura[#aktualnyNumerReceptury].Krok[#aktualnyKrokMycia].PM[15]
	                
	            THEN
	                "Cip".obiekt["Cip".tor[2].przepływomierzZaWymiennikiem].zerujLicznik1 := 0;
	                "Cip".obiekt["Cip".tor[2].przepływomierzZaWymiennikiem].startLicznik1 := 1;
	            ELSE
	                "Cip".obiekt["Cip".tor[2].przepływomierzZaWymiennikiem].startLicznik1 := 0;
	            END_IF;
	            
	            IF "Cip".obiekt["Cip".tor[2].przepływomierzZaWymiennikiem].licznik1 >
	                "Tor2_RecepturyStacjaMycia".Receptura[#aktualnyNumerReceptury].Krok[#aktualnyKrokMycia].PM[5]
	            THEN
	                "Cip".obiekt["Cip".tor[2].przepływomierzZaWymiennikiem].zerujLicznik1 := 0;
	                "Cip".obiekt["Cip".tor[2].przepływomierzZaWymiennikiem].startLicznik1 := 0;
	                "Cip".obiekt["Cip".tor[2].przepływomierzZaWymiennikiem].licznik1 := 0;
	                "Tor2_program".program.numerKroku := 7450;
	              
	            END_IF;
	            
	            
	            "Tor2_program".program.zadana1 := "Tor2_RecepturyStacjaMycia".Receptura[#aktualnyNumerReceptury].Krok[#aktualnyKrokMycia].PM[12] +
	            "Tor2_RecepturyStacjaMycia".Receptura[#aktualnyNumerReceptury].Krok[#aktualnyKrokMycia].PM[15];
	            "Tor2_program".program.aktualna1 := "Cip".obiekt["Cip".tor[2].przewodnośćNaPowrocie].WartośćPomiaru;
	            "Tor2_program".program.zadana2 := "Tor2_RecepturyStacjaMycia".Receptura[#aktualnyNumerReceptury].Krok[#aktualnyKrokMycia].PM[5];
	            "Tor2_program".program.aktualna2 := "Cip".obiekt["Cip".tor[2].przepływomierzZaWymiennikiem].licznik1;
	            
	            7450:// Drenaż zbiornika kwasu
	                
	                IF
	                    "Cip".obiekt["Cip".tor[2].czujnikPrzepływuNaPowrocie].hmiPotwWysterowania = 1
	                THEN
	                    "Tor2_program".program.opóżnienie := 0;
	                END_IF;
	                "IdźDoKroku"(inNumerKrokuDocelowy := 7460,
	                             inZadaneOpóżnienie   := "Tor2_RecepturyStacjaMycia".Receptura[#aktualnyNumerReceptury].Krok[#aktualnyKrokMycia].PM[7],
	                             numerKroku           := "Tor2_program".program.numerKroku,
	                             opóźnienie           := "Tor2_program".program.opóżnienie,
	                             pauza:=  "Tor2_hmi".button.bPauza.set);
	                
	                "Tor2_program".program.zadana1 := "Tor2_RecepturyStacjaMycia".Receptura[#aktualnyNumerReceptury].Krok[#aktualnyKrokMycia].PM[7];
	                "Tor2_program".program.aktualna1 := "Tor2_program".program.opóżnienie;
	                "Tor2_program".program.zadana2 := 0;
	                "Tor2_program".program.aktualna2 := INT_TO_REAL(BOOL_TO_INT("Cip".obiekt["Cip".tor[2].czujnikPrzepływuNaPowrocie].hmiPotwWysterowania = 1)) * 1.0;
	                
	            7460://     Płukanie główne zbiornika kwasu
	                
	                IF "Tor2_RecepturyStacjaMycia".Receptura[#aktualnyNumerReceptury].Krok[#aktualnyKrokMycia].PM[2] = 0
	                THEN
	                    ;
	                    "Tor2_program".program.numerKroku := 7470;
	                END_IF;
	                
	                
	                ;
	                IF "Cip".obiekt["Cip".tor[2].przewodnośćNaPowrocie].WartośćPomiaru <=
	                    "Tor2_RecepturyStacjaMycia".Receptura[#aktualnyNumerReceptury].Krok[#aktualnyKrokMycia].PM[12] +
	                    "Tor2_RecepturyStacjaMycia".Receptura[#aktualnyNumerReceptury].Krok[#aktualnyKrokMycia].PM[15]
	                  
	                THEN
	                    "Cip".obiekt["Cip".tor[2].przepływomierzZaWymiennikiem].zerujLicznik1 := 0;
	                    "Cip".obiekt["Cip".tor[2].przepływomierzZaWymiennikiem].startLicznik1 := 1;
	                ELSE
	                    "Cip".obiekt["Cip".tor[2].przepływomierzZaWymiennikiem].startLicznik1 := 0;
	                END_IF;
	                
	                IF "Cip".obiekt["Cip".tor[2].przepływomierzZaWymiennikiem].licznik1 >
	                    "Tor2_RecepturyStacjaMycia".Receptura[#aktualnyNumerReceptury].Krok[#aktualnyKrokMycia].PM[5]
	                THEN
	                    "Cip".obiekt["Cip".tor[2].przepływomierzZaWymiennikiem].zerujLicznik1 := 0;
	                    "Cip".obiekt["Cip".tor[2].przepływomierzZaWymiennikiem].startLicznik1 := 0;
	                    "Cip".obiekt["Cip".tor[2].przepływomierzZaWymiennikiem].licznik1 := 0;
	                    "Tor2_program".program.numerKroku := 7470;
	                 
	                 
	                END_IF;
	                
	                
	                "Tor2_program".program.zadana1 := "Tor2_RecepturyStacjaMycia".Receptura[#aktualnyNumerReceptury].Krok[#aktualnyKrokMycia].PM[12]+
	                "Tor2_RecepturyStacjaMycia".Receptura[#aktualnyNumerReceptury].Krok[#aktualnyKrokMycia].PM[15];
	                "Tor2_program".program.aktualna1 := "Cip".obiekt["Cip".tor[2].przewodnośćNaPowrocie].WartośćPomiaru;
	                "Tor2_program".program.zadana2 := "Tor2_RecepturyStacjaMycia".Receptura[#aktualnyNumerReceptury].Krok[#aktualnyKrokMycia].PM[5];
	                "Tor2_program".program.aktualna2 := "Cip".obiekt["Cip".tor[2].przepływomierzZaWymiennikiem].licznik1;
	                
	                7470:// Drenaż zbiornika kwasu
	                    
	                    IF
	                        "Cip".obiekt["Cip".tor[2].czujnikPrzepływuNaPowrocie].hmiPotwWysterowania = 1
	                    THEN
	                        "Tor2_program".program.opóżnienie := 0;
	                    END_IF;
	                    "IdźDoKroku"(inNumerKrokuDocelowy := 7290,
	                                 inZadaneOpóżnienie   := "Tor2_RecepturyStacjaMycia".Receptura[#aktualnyNumerReceptury].Krok[#aktualnyKrokMycia].PM[7],
	                                 numerKroku           := "Tor2_program".program.numerKroku,
	                                 opóźnienie           := "Tor2_program".program.opóżnienie,
	                                 pauza:=  "Tor2_hmi".button.bPauza.set);
	                    
	                    "Tor2_program".program.zadana1 := "Tor2_RecepturyStacjaMycia".Receptura[#aktualnyNumerReceptury].Krok[#aktualnyKrokMycia].PM[7];
	                    "Tor2_program".program.aktualna1 := "Tor2_program".program.opóżnienie;
	                    "Tor2_program".program.zadana2 := 0;
	                    "Tor2_program".program.aktualna2 := INT_TO_REAL(BOOL_TO_INT("Cip".obiekt["Cip".tor[2].czujnikPrzepływuNaPowrocie].hmiPotwWysterowania = 1)) * 1.0;
	           
	                    
	                7700://pauza
	                    "krokZapauzowany" := "krokZapauzowany";
	                        // IF "CIP1_hmi".button.bStart.set = 1 THEN
	                        //     "CIP1_program".program.numerKroku :="krokZapauzowany";//tu stary numer kroku
	                        // END_IF;
	                        IF "Tor2_hmi".button.bPauza.set = 0 THEN
	                            "Tor2_program".program.numerKroku := "krokZapauzowany";
	                        END_IF;
	                            ;
	                       
	                                
	                    END_CASE;
	                    //wejscie w pauze
	                    //
	            
	                    
	                            
	                            IF "Tor2_program".program.numerKroku <> 7700 THEN
	                                "krokZapauzowany" := "Tor2_program".program.numerKroku;
	                            END_IF;
	                            IF "Tor2_hmi".button.bPauza.set = 1 THEN
	                                
	                                "Tor2_program".program.numerKroku := 7700;
	                            END_IF;
END_FUNCTION

FUNCTION "Tor2.procedury_alarmow" : Void
{ S7_Optimized_Access := 'TRUE' }
VERSION : 0.1
   VAR_TEMP 
      obj : Int;
      nr : Int;
      Mnr : String;
      aktualnyNumerReceptury : Int;
      aktualnyKrokMycia : Int;
      nrSygnału : Int;
   END_VAR


BEGIN
	  //   //program zawiera procedury dla alarmow dla procedur o numerze >1  (procedura 0 i 1 jest obsługiwana w programie Obsługa alarmow)
	  //   //procedury wyzwalane  z progrmu TablicaProcedór dla kolejnych kroków  "F1".obiekt["F100CP01"].procedura: = 2
	  //   //wyzwolenie procedury zero  automatycznie  wyłącza alarm
	  //   //procedura:=1   uruchamia alarm
	  //   //
	  //   //open ctrl+shift+(*)Numeric
	  //   //close ctrl+shift+(/)Numeric
	  //   #aktualnyNumerReceptury := "CIP1_RecepturyStacjaMycia".numerUżywanejReceptury;
	  //   #aktualnyNumerReceptury := "CIP1_RecepturyStacjaMycia".numerUżywanejReceptury;
	  //   #aktualnyKrokMycia := "CIP1_RecepturyStacjaMycia".numerKrokuMycia;
	    
	  //   //alarmy
	  //   //
	  //   "Start_trig"(CLK:="CIP1_hmi".button.bStart.set =1);
	    
	  //   IF "Start_trig".Q =1 THEN
	  //       FOR "x" := 1 TO 14 DO
	  //           "CIP1_alarmy".alarm["x"].stan := 0;
	  //           "CIP1_alarmy".alarm["x"].timerek := 0;
	  //       END_FOR;
	  //   END_IF;
	  //   "CIP1_alarmy".alarm[14].stan := BOOL_TO_INT(NOT "diKSB_1");
	    
	  //   //Brak wody wtórnej
	    
	  //   #nr := 1;
	  //   CASE "CIP1_alarmy".alarm[#nr].procedura OF
	            
	  //       2: //zalacz
	  //           IF "CIP0_obiekty".obiekt["C1R1LL01"].hmiPotwWysterowania = 0
	  //               AND "CIP1_program".program.numerKroku >= 7210
	  //               AND "CIP1_program".program.numerKroku <= 7220
	                
	                
	                
	  //           THEN
	  //               IF "CIP1_alarmy".alarm[#nr].timerek < 32000 THEN
	  //                   "CIP1_alarmy".alarm[#nr].timerek := "CIP1_alarmy".alarm[#nr].timerek + 1;
	  //               END_IF;
	  //               "CIP1_alarmy".alarm[#nr].stan := BOOL_TO_INT("CIP1_alarmy".alarm[#nr].timerek > 100);
	  //           ELSE
	  //               "CIP1_alarmy".alarm[#nr].timerek := 0;
	  //               "CIP1_alarmy".alarm[#nr].stan := 0;
	  //           END_IF;
	            
	  //   END_CASE;
	    
	  //   // //Brak wody studziennej
	    
	  //   #nr := 2;
	  //   CASE "CIP1_alarmy".alarm[#nr].procedura OF
	            
	  //       2: //zalacz
	  //           IF "CIP1_obiekty".obiekt["C131LL11"].hmiPotwWysterowania = 0
	                
	                
	                
	  //           THEN
	  //               IF "CIP1_alarmy".alarm[#nr].timerek < 32000 THEN
	  //                   "CIP1_alarmy".alarm[#nr].timerek := "CIP1_alarmy".alarm[#nr].timerek + 1;
	  //               END_IF;
	  //               "CIP1_alarmy".alarm[#nr].stan := BOOL_TO_INT("CIP1_alarmy".alarm[#nr].timerek > 100);
	  //           ELSE
	  //               "CIP1_alarmy".alarm[#nr].timerek := 0;
	  //               "CIP1_alarmy".alarm[#nr].stan := 0;
	  //           END_IF;
	            
	  //           IF "CIP1_alarmy".alarm[#nr].stan = 1
	  //               AND "CIP1_program".program.numerKroku <> 7700 THEN
	  //               "CIP1_hmi".button.bPauza.set := 1;
	  //               "krokZapauzowany" := "CIP1_program".program.numerKroku;
	  //               "CIP1_program".program.numerKroku := 7700;
	  //           END_IF;
	            
	  //   END_CASE;
	    
	  //   //Brak ługu
	    
	  //   #nr := 3;
	  //   CASE "CIP1_alarmy".alarm[#nr].procedura OF
	            
	  //       2: //zalacz
	  //           IF "CIP0_obiekty".obiekt["C1L1LL01"].hmiPotwWysterowania = 0
	  //               AND #aktualnyKrokMycia = 3
	                
	                
	  //           THEN
	  //               IF "CIP1_alarmy".alarm[#nr].timerek < 32000 THEN
	  //                   "CIP1_alarmy".alarm[#nr].timerek := "CIP1_alarmy".alarm[#nr].timerek + 1;
	  //               END_IF;
	  //               "CIP1_alarmy".alarm[#nr].stan := BOOL_TO_INT("CIP1_alarmy".alarm[#nr].timerek > 100);
	  //           ELSE
	  //               "CIP1_alarmy".alarm[#nr].timerek := 0;
	  //               "CIP1_alarmy".alarm[#nr].stan := 0;
	  //           END_IF;
	            
	  //           IF "CIP1_alarmy".alarm[#nr].stan = 1
	  //               AND "CIP1_program".program.numerKroku <> 7700 THEN
	  //               "CIP1_hmi".button.bPauza.set := 1;
	  //               "krokZapauzowany" := "CIP1_program".program.numerKroku;
	  //               "CIP1_program".program.numerKroku := 7700;
	  //           END_IF;
	            
	  //   END_CASE;
	    
	  //   //Brak kwasu
	    
	  //   #nr := 4;
	  //   CASE "CIP1_alarmy".alarm[#nr].procedura OF
	            
	  //       2: //zalacz
	  //           IF "CIP0_obiekty".obiekt["C1A1LL01"].hmiPotwWysterowania = 0
	  //               AND #aktualnyKrokMycia = 4
	                
	                
	  //           THEN
	  //               IF "CIP1_alarmy".alarm[#nr].timerek < 32000 THEN
	  //                   "CIP1_alarmy".alarm[#nr].timerek := "CIP1_alarmy".alarm[#nr].timerek + 1;
	  //               END_IF;
	  //               "CIP1_alarmy".alarm[#nr].stan := BOOL_TO_INT("CIP1_alarmy".alarm[#nr].timerek > 100);
	  //           ELSE
	  //               "CIP1_alarmy".alarm[#nr].timerek := 0;
	  //               "CIP1_alarmy".alarm[#nr].stan := 0;
	  //           END_IF;
	            
	  //           IF "CIP1_alarmy".alarm[#nr].stan = 1
	  //               AND "CIP1_program".program.numerKroku <> 7700 THEN
	  //               "CIP1_hmi".button.bPauza.set := 1;
	  //               "krokZapauzowany" := "CIP1_program".program.numerKroku;
	  //               "CIP1_program".program.numerKroku := 7700;
	  //           END_IF;
	            
	  //   END_CASE;
	    
	  // //  Brak gotowości obiektu
	    
	  //   #nr := 5;
	  //   CASE "CIP1_alarmy".alarm[#nr].procedura OF
	            
	  //       2: //zalacz
	  //           #nrSygnału :=
	  //           REAL_TO_INT("CIP1_RecepturyStacjaMycia".Receptura[#aktualnyNumerReceptury].Krok[#aktualnyKrokMycia].PM[24]);
	  //           IF "CIP1_RecepturyStacjaMycia".Receptura[#aktualnyNumerReceptury].Krok[#aktualnyKrokMycia].PM[21]=1
	  //               AND
	  //               "SIG".SIG[#nrSygnału] = 0
	  //           THEN
	  //               IF "CIP1_alarmy".alarm[#nr].timerek < 32000 THEN
	  //                   "CIP1_alarmy".alarm[#nr].timerek := "CIP1_alarmy".alarm[#nr].timerek + 1;
	  //               END_IF;
	  //               "CIP1_alarmy".alarm[#nr].stan := BOOL_TO_INT("CIP1_alarmy".alarm[#nr].timerek > 50);
	  //           ELSE
	  //               "CIP1_alarmy".alarm[#nr].timerek := 0;
	  //               "CIP1_alarmy".alarm[#nr].stan := 0;
	  //           END_IF;
	            
	  //           IF "CIP1_alarmy".alarm[#nr].stan = 1
	  //               AND "CIP1_program".program.numerKroku <> 7700 THEN
	  //               "CIP1_hmi".button.bPauza.set := 1;
	  //               "krokZapauzowany" := "CIP1_program".program.numerKroku;
	  //               "CIP1_program".program.numerKroku := 7700;
	  //           END_IF;
	            
	  //   END_CASE;
	    
	    
	  //  // Brak przepływu na zasilaniu
	    
	  //   #nr := 6;
	  //   CASE "CIP1_alarmy".alarm[#nr].procedura OF
	            
	  //       2: //zalacz
	  //           IF "CIP1_obiekty".obiekt["C101FT11"].WartośćPomiaru <=
	  //               0.2*"CIP1_RecepturyStacjaMycia".Receptura[#aktualnyNumerReceptury].Krok[#aktualnyKrokMycia].PM[2]
	  //               AND "CIP1_obiekty".obiekt["C101CP11"].inZadaneWysterowanieAuto>10
	                
	  //           THEN
	  //               IF "CIP1_alarmy".alarm[#nr].timerek < 32000
	  //                   AND "CIP1_obiekty".obiekt[1].outStartUrządzenie AND ("CIP1_hmi".button.bPauza.set=0)
	  //               THEN
	  //                   "CIP1_alarmy".alarm[#nr].timerek := "CIP1_alarmy".alarm[#nr].timerek + 1;
	  //               END_IF;
	  //               "CIP1_alarmy".alarm[#nr].stan := BOOL_TO_INT("CIP1_alarmy".alarm[#nr].timerek >
	  //               "CIP1_RecepturyStacjaMycia".Receptura[#aktualnyNumerReceptury].Krok[#aktualnyKrokMycia].PM[3]*10);
	  //           ELSE
	  //               "CIP1_alarmy".alarm[#nr].timerek := 0;
	  //               "CIP1_alarmy".alarm[#nr].stan := 0;
	  //           END_IF;
	            
	  //           IF "CIP1_alarmy".alarm[#nr].stan = 1
	  //               AND "CIP1_program".program.numerKroku <> 7700 THEN
	  //               "CIP1_hmi".button.bPauza.set := 1;
	  //               "krokZapauzowany" := "CIP1_program".program.numerKroku;
	  //               "CIP1_program".program.numerKroku := 7700;
	  //           END_IF;
	            
	  //         0:
	  //             "CIP1_alarmy".alarm[#nr].timerek := 0;
	  //             "CIP1_alarmy".alarm[#nr].stan := 0;
	              
	            
	  //   END_CASE;
	    
	  //   IF "CIP1_obiekty".obiekt["C101CP11"].inZadaneWysterowanieAuto < 10 THEN
	  //       "CIP1_alarmy".alarm[#nr].timerek := 0;
	  //       "CIP1_alarmy".alarm[#nr].stan := 0;
	  //   END_IF;
	    
	  //  // Brak przepływu na powrocie
	    
	  //   #nr := 7;
	  //   CASE "CIP1_alarmy".alarm[#nr].procedura OF
	            
	  //       2: //zalacz
	  //           IF "CIP1_obiekty".obiekt["C101FV11"].hmiPotwWysterowania =0 AND ("CIP1_hmi".button.bPauza.set=0)
	                
	                
	  //           THEN
	  //               IF "CIP1_alarmy".alarm[#nr].timerek < 32000 THEN
	  //                   "CIP1_alarmy".alarm[#nr].timerek := "CIP1_alarmy".alarm[#nr].timerek + 1;
	  //               END_IF;
	  //               "CIP1_alarmy".alarm[#nr].stan := BOOL_TO_INT("CIP1_alarmy".alarm[#nr].timerek >
	  //               "CIP1_RecepturyStacjaMycia".Receptura[#aktualnyNumerReceptury].Krok[#aktualnyKrokMycia].PM[4] * 10);
	  //           ELSE
	  //               "CIP1_alarmy".alarm[#nr].timerek := 0;
	  //               "CIP1_alarmy".alarm[#nr].stan := 0;
	  //           END_IF;
	            
	  //           IF "CIP1_alarmy".alarm[#nr].stan = 1
	  //               AND "CIP1_program".program.numerKroku <> 7700 THEN
	  //               "CIP1_hmi".button.bPauza.set := 1;
	  //               "krokZapauzowany" := "CIP1_program".program.numerKroku;
	  //               "CIP1_program".program.numerKroku := 7700;
	  //           END_IF;
	            
	  //       0:
	  //           "CIP1_alarmy".alarm[#nr].timerek := 0;
	  //           "CIP1_alarmy".alarm[#nr].stan := 0;
	            
	  //   END_CASE;
	    
	    
	    
	  //   //Niskie stężenie ługu
	    
	  //   #nr :=8;
	  //   CASE "CIP1_alarmy".alarm[#nr].procedura OF
	            
	  //       2: //zalacz
	  //           IF "CIP1_obiekty".obiekt["C101CT11"].WartośćPomiaru <=
	  //               0.5 * "CIP1_RecepturyStacjaMycia".Receptura[#aktualnyNumerReceptury].Krok[#aktualnyKrokMycia].PM[10]
	  //               AND #aktualnyKrokMycia=3
	                
	  //           THEN
	  //               IF "CIP1_alarmy".alarm[#nr].timerek < 32000 THEN
	  //                   "CIP1_alarmy".alarm[#nr].timerek := "CIP1_alarmy".alarm[#nr].timerek + 1;
	  //               END_IF;
	  //               "CIP1_alarmy".alarm[#nr].stan := BOOL_TO_INT("CIP1_alarmy".alarm[#nr].timerek >600);
	  //           ELSE
	  //               "CIP1_alarmy".alarm[#nr].timerek := 0;
	  //               "CIP1_alarmy".alarm[#nr].stan := 0;
	  //           END_IF;
	        
	            
	  //   END_CASE;
	    
	    
	    
	    
	  //   //Niskie stężenie kwasu
	    
	  //   #nr := 9;
	  //   CASE "CIP1_alarmy".alarm[#nr].procedura OF
	            
	  //       2: //zalacz
	  //           IF "CIP1_obiekty".obiekt["C101CT11"].WartośćPomiaru <=
	  //               0.5 * "CIP1_RecepturyStacjaMycia".Receptura[#aktualnyNumerReceptury].Krok[#aktualnyKrokMycia].PM[10]
	  //               AND #aktualnyKrokMycia=4
	                
	  //           THEN
	  //               IF "CIP1_alarmy".alarm[#nr].timerek < 32000 THEN
	  //                   "CIP1_alarmy".alarm[#nr].timerek := "CIP1_alarmy".alarm[#nr].timerek + 1;
	  //               END_IF;
	  //               "CIP1_alarmy".alarm[#nr].stan := BOOL_TO_INT("CIP1_alarmy".alarm[#nr].timerek > 600);
	  //           ELSE
	  //               "CIP1_alarmy".alarm[#nr].timerek := 0;
	  //               "CIP1_alarmy".alarm[#nr].stan := 0;
	  //           END_IF;
	            
	       
	            
	  //   END_CASE;
	    
	    
	  //   //Brak stężonego ługu
	    
	  //   #nr := 10;
	  //   CASE "CIP1_alarmy".alarm[#nr].procedura OF
	            
	  //       2: //zalacz
	  //           IF "CIP0_obiekty".obiekt["C2L1LL01"].hmiPotwWysterowania = 0
	                
	                
	                
	  //           THEN
	  //               IF "CIP1_alarmy".alarm[#nr].timerek < 32000 THEN
	  //                   "CIP1_alarmy".alarm[#nr].timerek := "CIP1_alarmy".alarm[#nr].timerek + 1;
	  //               END_IF;
	  //               "CIP1_alarmy".alarm[#nr].stan := BOOL_TO_INT("CIP1_alarmy".alarm[#nr].timerek > 600);
	  //           ELSE
	  //               "CIP1_alarmy".alarm[#nr].timerek := 0;
	  //               "CIP1_alarmy".alarm[#nr].stan := 0;
	  //           END_IF;
	            
	          
	            
	  //   END_CASE;
	    
	  //   //Brak stężonego kwasu
	    
	  //   #nr := 11;
	  //   CASE "CIP1_alarmy".alarm[#nr].procedura OF
	            
	  //       2: //zalacz
	  //           IF "CIP0_obiekty".obiekt["C2A1LL01"].hmiPotwWysterowania = 0
	                
	                
	                
	  //           THEN
	  //               IF "CIP1_alarmy".alarm[#nr].timerek < 32000 THEN
	  //                   "CIP1_alarmy".alarm[#nr].timerek := "CIP1_alarmy".alarm[#nr].timerek + 1;
	  //               END_IF;
	  //               "CIP1_alarmy".alarm[#nr].stan := BOOL_TO_INT("CIP1_alarmy".alarm[#nr].timerek > 600);
	  //           ELSE
	  //               "CIP1_alarmy".alarm[#nr].timerek := 0;
	  //               "CIP1_alarmy".alarm[#nr].stan := 0;
	  //           END_IF;
	    
	            
	  //   END_CASE;
	    
	  //   //Brak dezynfekanta
	    
	  //   #nr := 12;
	  //   CASE "CIP1_alarmy".alarm[#nr].procedura OF
	            
	  //       2: //zalacz
	  //           IF "CIP0_obiekty".obiekt["C2D1LL01"].hmiPotwWysterowania = 0
	                
	                
	                
	  //           THEN
	  //               IF "CIP1_alarmy".alarm[#nr].timerek < 32000 THEN
	  //                   "CIP1_alarmy".alarm[#nr].timerek := "CIP1_alarmy".alarm[#nr].timerek + 1;
	  //               END_IF;
	  //               "CIP1_alarmy".alarm[#nr].stan := BOOL_TO_INT("CIP1_alarmy".alarm[#nr].timerek > 600);
	  //           ELSE
	  //               "CIP1_alarmy".alarm[#nr].timerek := 0;
	  //               "CIP1_alarmy".alarm[#nr].stan := 0;
	  //           END_IF;
	         
	  //   END_CASE;
	    
	    
	        
	  //       #nr := 13;
	  //       CASE "CIP1_alarmy".alarm[#nr].procedura OF
	                
	  //           2: //zalacz
	  //               IF  "CIP1_program".program.opóżnienie
	  //                   >"CIP1_RecepturyStacjaMycia".Receptura[#aktualnyNumerReceptury].Krok[#aktualnyKrokMycia].PM[19]
	                    
	                    
	  //               THEN
	  //                   IF "CIP1_alarmy".alarm[#nr].timerek < 32000 THEN
	  //                       "CIP1_alarmy".alarm[#nr].timerek := "CIP1_alarmy".alarm[#nr].timerek + 1;
	  //                   END_IF;
	  //                   "CIP1_alarmy".alarm[#nr].stan := BOOL_TO_INT("CIP1_alarmy".alarm[#nr].timerek > 600);
	  //               ELSE
	  //                   "CIP1_alarmy".alarm[#nr].timerek := 0;
	  //                   "CIP1_alarmy".alarm[#nr].stan := 0;
	  //               END_IF;
	         
	                
	  //       END_CASE;
	  
END_FUNCTION

FUNCTION "Tor2.procedury_obiektów" : Void
{ S7_Optimized_Access := 'TRUE' }
VERSION : 0.1
   VAR_TEMP 
      obj : Int;
      nr : Int;
      Mnr : String;
      aktualnyNumerReceptury : Int;
      aktualnyKrokMycia : Int;
      temp : Int;
   END_VAR


BEGIN
	    //program zawiera procedury dla napedów i zaworów dla procedur o numerze >1  (procedura 0 i 1 jest obsługiwana w programie Obsługa obiektów)
	    //procedury wyzwalane  z progrmu TablicaProcedór dla kolejnych kroków  "F1".obiekt["F100CP01"].procedura: = 2
	    //wyzwolenie procedury zero  automatycznie  wyłącza naped/zawór
	    //procedura:=1   uruchamia napęd/zawór na 100% - czyli załaczenie napedu jak kiedyś SET -- obsługiwana jest w programie Obsługa obiektów
	    //PAUZA może być obsługiwana w każdej procedurze z osobna
	    //
	    //open ctrl+shift+(*)Numeric
	    //close ctrl+shift+(/)Numeric
	    
	    #aktualnyNumerReceptury := "Tor2_RecepturyStacjaMycia".numerUżywanejReceptury;
	    #aktualnyKrokMycia := "Tor2_RecepturyStacjaMycia".numerKrokuMycia;
	    #temp := "Tor2_program".program.numerKroku;
	    
	    REGION POMPA PODAWANIA CIP
	    
	        #nr := "Cip".tor[2].pompaPodawaniaCip;
	    CASE "Tor2_program".program.numerKroku OF
	    7210, 7220, 7250:
	    "Cip".obiekt[#nr].procedura := 2;
	7244, 7270, 7281..7287, 7285, 7287,7310,7320, 7321, 7414, 7420:
	    "Cip".obiekt[#nr].procedura := 3;
	    7240, 7242, 7243, 7246:
	    "Cip".obiekt[#nr].procedura := 6;
	    7100:
	    "Cip".obiekt[#nr].procedura := 7;
	    ELSE
	    "Cip".obiekt[#nr].procedura := 0;
	    
	    END_CASE;
	    
	    
	    
	    CASE "Cip".obiekt[#nr].procedura OF
	    2:
	    //wyzwolenie timerków
	    "Cip".obiekt[#nr].SetReset.czasDoSet := 3;
	    "Cip".obiekt[#nr].SetReset.inSet := "Cip".obiekt["Cip".tor[0].zbiornikwodyCzystej.czujnikDolnegoPoziomu].hmiPotwWysterowania
	    OR "Cip".obiekt["Cip".tor[0].zbiornikWodyWtórnej.czujnikDolnegoPoziomu].hmiPotwWysterowania;
	    "Cip".obiekt[#nr].SetReset.czasDoReset := 5;
	    "Cip".obiekt[#nr].SetReset.inReset := (NOT "Cip".obiekt["Cip".tor[0].zbiornikwodyCzystej.czujnikDolnegoPoziomu].hmiPotwWysterowania
	    AND NOT "Cip".obiekt["Cip".tor[0].zbiornikWodyWtórnej.czujnikDolnegoPoziomu].hmiPotwWysterowania) OR
	    ("Cip".obiekt["Cip".tor[1].zbiornikDezynfekantu.czujnikDolnegoPoziomu].hmiPotwWysterowania = 0 AND ("Tor1_program".program.numerKroku = 7282
	    OR "Tor1_program".program.numerKroku = 7283));
	    
	    //załaczanie
	    "Cip".obiekt[#nr].inStartAuto := "Cip".obiekt[#nr].SetReset.wyjście;
	    
	    //wysterowanie
	    "Cip".obiekt[#nr].inZadaneWysterowanieAuto :=  //pid_out wypełniamy w wywołaniu pida z out pida
	    LIMIT(IN := "Cip".obiekt[#nr].pid_Out, MN := 0.0, MX := 100.0);//pid_out ;
	    
	    ////PID
	    "Cip".obiekt[#nr].pid_SP := "Tor2_RecepturyStacjaMycia".Receptura[#aktualnyNumerReceptury].Krok[#aktualnyKrokMycia].PM[2];
	    "Cip".obiekt[#nr].pid_PV := "Cip".obiekt["Cip".tor[2].przepływomierzZaWymiennikiem].WartośćPomiaru;
	    
	    
	    3: //wyzwolenie timerków
	    
	    //wyzwolenie timerków
	    "Cip".obiekt[#nr].SetReset.czasDoSet := 3;
	    "Cip".obiekt[#nr].SetReset.inSet := "Cip".obiekt["Cip".tor[0].zbiornikwodyCzystej.czujnikDolnegoPoziomu].hmiPotwWysterowania
	    ;
	    "Cip".obiekt[#nr].SetReset.czasDoReset := 5;
	    "Cip".obiekt[#nr].SetReset.inReset := NOT "Cip".obiekt["Cip".tor[0].zbiornikwodyCzystej.czujnikDolnegoPoziomu].hmiPotwWysterowania
	    ;
	    //załaczanie
	    
	    "Cip".obiekt[#nr].inStartAuto := "Cip".obiekt[#nr].SetReset.wyjście;
	    
	    //wysterowanie
	    "Cip".obiekt[#nr].inZadaneWysterowanieAuto :=  //pid_out wypełniamy w wywołaniu pida z out pida
	    LIMIT(IN := "Cip".obiekt[#nr].pid_Out, MN := 0.0, MX := 100.0);//pid_out ;
	    
	    ////PID
	    "Cip".obiekt[#nr].pid_SP := "Tor2_RecepturyStacjaMycia".Receptura[#aktualnyNumerReceptury].Krok[#aktualnyKrokMycia].PM[2];
	    "Cip".obiekt[#nr].pid_PV := "Cip".obiekt["Cip".tor[2].przepływomierzZaWymiennikiem].WartośćPomiaru;
	    
	    4: //wyzwolenie timerków
	    
	    //wyzwolenie timerków
	    "Cip".obiekt[#nr].SetReset.czasDoSet := 3;
	    "Cip".obiekt[#nr].SetReset.inSet :=
	    "Cip".obiekt["Cip".tor[0].zbiornikwodyCzystej.czujnikDolnegoPoziomu].hmiPotwWysterowania
	    AND #aktualnyKrokMycia = 3
	    ;
	    "Cip".obiekt[#nr].SetReset.czasDoReset := 5;
	    "Cip".obiekt[#nr].SetReset.inReset :=
	    NOT "Cip".obiekt["Cip".tor[0].zbiornikwodyCzystej.czujnikDolnegoPoziomu].hmiPotwWysterowania
	    AND #aktualnyKrokMycia = 3
	    ;
	    //załaczanie
	    "Cip".obiekt[#nr].inStartAuto := "Cip".obiekt[#nr].SetReset.wyjście;
	    
	    //wysterowanie
	    "Cip".obiekt[#nr].inZadaneWysterowanieAuto :=  //pid_out wypełniamy w wywołaniu pida z out pida
	    LIMIT(IN := "Cip".obiekt[#nr].pid_Out, MN := 0.0, MX := 100.0);//pid_out ;
	    
	    ////PID
	    "Cip".obiekt[#nr].pid_SP := "Tor2_RecepturyStacjaMycia".Receptura[#aktualnyNumerReceptury].Krok[#aktualnyKrokMycia].PM[2];
	    "Cip".obiekt[#nr].pid_PV := "Cip".obiekt["Cip".tor[2].przepływomierzZaWymiennikiem].WartośćPomiaru;
	    
	    5: //wyzwolenie timerków
	    
	    //wyzwolenie timerków
	    "Cip".obiekt[#nr].SetReset.czasDoSet := 3;
	    "Cip".obiekt[#nr].SetReset.inSet := "Cip".obiekt["Cip".tor[0].zbiornikwodyCzystej.czujnikDolnegoPoziomu].hmiPotwWysterowania
	    AND #aktualnyKrokMycia = 4
	    ;
	    "Cip".obiekt[#nr].SetReset.czasDoReset := 5;
	    "Cip".obiekt[#nr].SetReset.inReset := NOT "Cip".obiekt["Cip".tor[0].zbiornikwodyCzystej.czujnikDolnegoPoziomu].hmiPotwWysterowania
	    AND #aktualnyKrokMycia = 4
	    ;
	    //załaczanie
	    "Cip".obiekt[#nr].inStartAuto := "Cip".obiekt[#nr].SetReset.wyjście;
	    
	    //wysterowanie
	    "Cip".obiekt[#nr].inZadaneWysterowanieAuto :=  //pid_out wypełniamy w wywołaniu pida z out pida
	    LIMIT(IN := "Cip".obiekt[#nr].pid_Out, MN := 0.0, MX := 100.0);//pid_out ;
	    
	    ////PID
	    "Cip".obiekt[#nr].pid_SP := "Tor2_RecepturyStacjaMycia".Receptura[#aktualnyNumerReceptury].Krok[#aktualnyKrokMycia].PM[2];
	    "Cip".obiekt[#nr].pid_PV := "Cip".obiekt["Cip".tor[2].przepływomierzZaWymiennikiem].WartośćPomiaru;
	    
	    6: //wyzwolenie timerków
	    //wyzwolenie timerków
	    "Cip".obiekt[#nr].SetReset.czasDoSet := 3;
	    "Cip".obiekt[#nr].SetReset.inSet :=
	    ("Cip".obiekt["Cip".tor[0].zbiornikwodyCzystej.czujnikDolnegoPoziomu].hmiPotwWysterowania
	    AND #aktualnyKrokMycia = 4)
	    OR
	    ("Cip".obiekt["Cip".tor[0].zbiornikwodyCzystej.czujnikDolnegoPoziomu].hmiPotwWysterowania
	    AND #aktualnyKrokMycia = 3)
	    ;
	    "Cip".obiekt[#nr].SetReset.czasDoReset := 5;
	    "Cip".obiekt[#nr].SetReset.inReset :=
	    (NOT "Cip".obiekt["Cip".tor[0].zbiornikwodyCzystej.czujnikDolnegoPoziomu].hmiPotwWysterowania
	    AND #aktualnyKrokMycia = 4)
	    OR
	    (NOT "Cip".obiekt["Cip".tor[0].zbiornikwodyCzystej.czujnikDolnegoPoziomu].hmiPotwWysterowania
	    AND #aktualnyKrokMycia = 3);
	    
	    //załaczanie
	    "Cip".obiekt[#nr].inStartAuto := 1;
	    
	    //wysterowanie
	    "Cip".obiekt[#nr].inZadaneWysterowanieAuto :=  //pid_out wypełniamy w wywołaniu pida z out pida
	    LIMIT(IN := "Cip".obiekt[#nr].pid_Out, MN := 0.0, MX := 100.0);//pid_out ;
	    
	    ////PID
	    "Cip".obiekt[#nr].pid_SP := "Tor2_RecepturyStacjaMycia".Receptura[#aktualnyNumerReceptury].Krok[#aktualnyKrokMycia].PM[2];
	    "Cip".obiekt[#nr].pid_PV := "Cip".obiekt["Cip".tor[2].przepływomierzZaWymiennikiem].WartośćPomiaru;
	    
	    
	    7:
	    //wyzwolenie timerków
	    "Cip".obiekt[#nr].SetReset.czasDoSet := 1;
	    "Cip".obiekt[#nr].SetReset.inSet :=
	    "Cip".obiekt["Cip".tor[2].pompaPodawaniaCip].inStartAuto; //cpNiex
	    
	    "Cip".obiekt[#nr].SetReset.czasDoReset := 1;
	    "Cip".obiekt[#nr].SetReset.inReset :=
	    NOT "Cip".obiekt["Cip".tor[2].pompaPodawaniaCip].inStartAuto; //cpNiex
	    //załaczanie
	    "Cip".obiekt[#nr].inStartAuto := "Cip".obiekt[#nr].SetReset.wyjście;
	    //wysterowanie
	    "Cip".obiekt[#nr].inZadaneWysterowanieAuto := 100.0;
	    
	    
	    
	    0:
	    ;
	    
	    // resetowanie całkującej części regulatora aby nie przejebać temperatury
	    // "PID_Compact23".IntegralResetMode := 3;
	    // "PID_Compact23".OverwriteInitialOutputValue := "F1.SP"."203"- 1.0;
	    // "PID_Compact23".Reset := "F1".obiekt["F100LT01"].WartośćPomiaru > 70.0;
	    // := LIMIT(IN := "APA".obiekt["PID123"].outWysterowanieUrządzenia,
	    // MN := 0.0, MX := "APA".obiekt["H101TT01"].WartośćPomiaru + "H1.STP"."214");
	    
	    END_CASE;
	    
	    IF "Cip".obiekt[#nr].procedura > 0 THEN
	    
	    IF "Cip".obiekt[#nr].inStartAuto = 0 THEN
	    "Cip".obiekt[#nr].inZadaneWysterowanieAuto := 0.0;
	    "Cip".obiekt[#nr].pid_SP := 0.0;
	    END_IF;
	    END_IF;
	    
	    
	    "PID.pompaPodawaniaCipTor1"(Setpoint := "Cip".obiekt[#nr].pid_SP,
	                        Input := "Cip".obiekt[#nr].pid_PV,
	                        Reset := "Cip".obiekt[#nr].hmiResetAwaria,
	                        Output => "Cip".obiekt[#nr].pid_Out);
	    "PID.pompaPodawaniaCipTor1".Retain.CtrlParams.Gain := 1.2;
	    "PID.pompaPodawaniaCipTor1".Retain.CtrlParams.Ti := 3;
	    "PID.pompaPodawaniaCipTor1".Retain.CtrlParams.Td := 0.2;
	    
	    
	    
	    "PID.pompaPodawaniaCipTor1".IntegralResetMode := 3;
	    "PID.pompaPodawaniaCipTor1".OverwriteInitialOutputValue := 1;
	    "PID.pompaPodawaniaCipTor1".Reset := (
	    "Cip".obiekt[#nr].procedura = 0 OR "Cip".obiekt[#nr].inStartAuto = 0
	    OR "numer_kroku_stary_2" <> "Tor2_program".program.numerKroku);
	    
	    "numer_kroku_stary_2" := "Tor2_program".program.numerKroku;
	    END_REGION
	    
	    REGION POMPA PRZYGOTOWANIA CIP(DRUGA PODAWCZA)
	    
	    //pompa powrotu/ Program musi ustalić, który tor myje stacje,
	    //drugi staje się pompą powrotu (staje się pompą 102 - tymczasowo)
	    //obsługa wykrywania w CIP1_wejściach_wyjściach
	    #nr := "Cip".tor[2].pompaPodawaniaCip;
	    CASE "Tor2_program".program.numerKroku OF
	    7401..7404, 7410..7414:
	    "Cip".obiekt[#nr].procedura := 2
	    ;
	    7230..7440:
	    "Cip".obiekt[#nr].procedura := 3;
	    7450, 7460:
	    "Cip".obiekt[#nr].procedura := 4;
	    ELSE
	    "Cip".obiekt[#nr].procedura := 0;
	    
	    END_CASE;
	    
	    
	    CASE "Cip".obiekt[#nr].procedura OF
	    2:
	    //wyzwolenie timerków
	    "Cip".obiekt[#nr].SetReset.czasDoSet := 3;
	    "Cip".obiekt[#nr].SetReset.inSet :=
	    "Cip".obiekt["Cip".tor[0].zbiornikWodyWtórnej.czujnikDolnegoPoziomu].hmiPotwWysterowania;
	    
	    "Cip".obiekt[#nr].SetReset.czasDoReset := 60;
	    "Cip".obiekt[#nr].SetReset.inReset :=
	    NOT "Cip".obiekt["Cip".tor[0].zbiornikWodyWtórnej.czujnikDolnegoPoziomu].hmiPotwWysterowania;
	    //załaczanie
	    
	    "Cip".obiekt[#nr].inStartAuto := "Cip".obiekt[#nr].SetReset.wyjście;
	    
	    //wysterowanie
	    "Cip".obiekt[#nr].inZadaneWysterowanieAuto := 100.0;
	    
	    3:
	    //wyzwolenie timerków
	    "Cip".obiekt[#nr].SetReset.czasDoSet := 3;
	    "Cip".obiekt[#nr].SetReset.inSet :=
	    "Cip".obiekt["Cip".tor[0].zbiornikŁugu.czujnikDolnegoPoziomu].hmiPotwWysterowania;
	    
	    "Cip".obiekt[#nr].SetReset.czasDoReset := 60;
	    "Cip".obiekt[#nr].SetReset.inReset :=
	    NOT "Cip".obiekt["Cip".tor[0].zbiornikŁugu.czujnikDolnegoPoziomu].hmiPotwWysterowania;
	    //załaczanie
	    
	    "Cip".obiekt[#nr].inStartAuto := "Cip".obiekt[#nr].SetReset.wyjście;
	    
	    //wysterowanie
	    "Cip".obiekt[#nr].inZadaneWysterowanieAuto := 100.0;
	    4:
	    //wyzwolenie timerków
	    "Cip".obiekt[#nr].SetReset.czasDoSet := 3;
	    "Cip".obiekt[#nr].SetReset.inSet :=
	    "Cip".obiekt["Cip".tor[0].zbiornikKwasu.czujnikDolnegoPoziomu].hmiPotwWysterowania;
	    
	    "Cip".obiekt[#nr].SetReset.czasDoReset := 60;
	    "Cip".obiekt[#nr].SetReset.inReset :=
	    NOT "Cip".obiekt["Cip".tor[0].zbiornikKwasu.czujnikDolnegoPoziomu].hmiPotwWysterowania;
	    //załaczanie
	    "Cip".obiekt[#nr].inStartAuto := "Cip".obiekt[#nr].SetReset.wyjście;
	    //wysterowanie
	    "Cip".obiekt[#nr].inZadaneWysterowanieAuto := 100.0;
	    
	    
	    
	    END_CASE;
	    
	    END_REGION
	    
	    REGION ZAWÓR DOZOWANIA ŁUGU W LINIE
	    
	        #nr := "Cip".tor[0].zawórDozowaniaLuguwLinię;
	        
	        CASE "Tor2_program".program.numerKroku OF
	            7243, 7320:
	                "Cip".obiekt[#nr].procedura := 3;
	            ELSE
	                "Cip".obiekt[#nr].procedura := 0;
	        END_CASE;
	        
	    CASE "Cip".obiekt[#nr].procedura OF
	    2:
	    //set - warunki dla wejścia funkcji Set
	    "Cip".obiekt[#nr].SetReset.czasDoSet := 10;
	    "Cip".obiekt[#nr].SetReset.inSet :=
	    "Cip".obiekt["Cip".tor[0].zbiorniczekDozowaniaŁugu.czujnikDolnegoPoziomu].hmiPotwWysterowania = 1
	    AND #aktualnyKrokMycia = 3;
	    
	    //reset - warunki dla wejścia funkcji Reset
	    "Cip".obiekt[#nr].SetReset.czasDoReset := 0;
	    "Cip".obiekt[#nr].SetReset.inReset :=
	    "Cip".obiekt["Cip".tor[0].zbiorniczekDozowaniaŁugu.czujnikDolnegoPoziomu].hmiPotwWysterowania = 0
	    OR #aktualnyKrokMycia = 4;
	    
	    //załaczanie
	    "Cip".obiekt[#nr].Flipaj.czas_ON := 300;
	    "Cip".obiekt[#nr].Flipaj.czas_OFF := 100;
	    "Cip".obiekt[#nr].Flipaj.ile_petli := 999;
	    "Cip".obiekt[#nr].Flipaj.in := "Cip".obiekt[#nr].SetReset.wyjście;
	    "Cip".obiekt[#nr].inStartAuto := "Cip".obiekt[#nr].Flipaj.Q;
	    
	    //wysterowanie
	    "Cip".obiekt[#nr].inZadaneWysterowanieAuto := 100.0;
	    
	    3:
	    //set - warunki dla wejścia funkcji Set
	    "Cip".obiekt[#nr].SetReset.czasDoSet := 10;
	    "Cip".obiekt[#nr].SetReset.inSet :=
	    "Cip".obiekt["Cip".tor[0].zbiorniczekDozowaniaŁugu.czujnikDolnegoPoziomu].hmiPotwWysterowania = 1
	    AND ("Tor2_RecepturyStacjaMycia".numerKrokuMycia = 3)
	    AND ("Cip".obiekt["Cip".tor[2].przewodnośćNaPowrocie].WartośćPomiaru <
	    "Tor2_RecepturyStacjaMycia".Receptura[#aktualnyNumerReceptury].Krok[#aktualnyKrokMycia].PM[11]);
	    
	    //reset - warunki dla wejścia funkcji Reset
	    "Cip".obiekt[#nr].SetReset.czasDoReset := 0;
	    "Cip".obiekt[#nr].SetReset.inReset :=
	    "Cip".obiekt["Cip".tor[0].zbiorniczekDozowaniaŁugu.czujnikDolnegoPoziomu].hmiPotwWysterowania = 0
	    OR ("Tor2_RecepturyStacjaMycia".numerKrokuMycia = 4)
	    OR ("Cip".obiekt["Cip".tor[2].przewodnośćNaPowrocie].WartośćPomiaru >=
	    "Tor2_RecepturyStacjaMycia".Receptura[#aktualnyNumerReceptury].Krok[#aktualnyKrokMycia].PM[11]);
	    
	    //załaczanie
	    "Cip".obiekt[#nr].Flipaj.czas_ON := REAL_TO_INT(
	                                                    "Tor2_RecepturyStacjaMycia".
	                                                    Receptura[#aktualnyNumerReceptury].
	                                                    Krok[#aktualnyKrokMycia].PM[26] * 10);
	    "Cip".obiekt[#nr].Flipaj.czas_OFF := REAL_TO_INT(
	                                                     "Tor2_RecepturyStacjaMycia".
	                                                     Receptura[#aktualnyNumerReceptury].
	                                                     Krok[#aktualnyKrokMycia].PM[27] * 10);
	    "Cip".obiekt[#nr].Flipaj.ile_petli :=
	    REAL_TO_INT("Tor2_RecepturyStacjaMycia".Receptura[#aktualnyNumerReceptury].Krok[#aktualnyKrokMycia].PM[20] /
	                ("Tor2_RecepturyStacjaMycia".Receptura[#aktualnyNumerReceptury].Krok[#aktualnyKrokMycia].PM[26] +
	                "Tor2_RecepturyStacjaMycia".Receptura[#aktualnyNumerReceptury].Krok[#aktualnyKrokMycia].PM[27] + 1.0));
	    "Cip".obiekt[#nr].Flipaj.in := "Cip".obiekt[#nr].SetReset.wyjście;
	    "Cip".obiekt[#nr].inStartAuto := "Cip".obiekt[#nr].Flipaj.Q;
	    
	    //wysterowanie
	    "Cip".obiekt[#nr].inZadaneWysterowanieAuto := 100.0;
	0:
	    "Cip".obiekt[#nr].Flipaj.in := 0;
	    END_CASE;
	    END_REGION
	    
	    REGION ZAWÓR DOZOWANIA KWASU W LINIE
	    
	        #nr := "Cip".tor[0].zawórDozowaniaKwasuwLinię;
	        
	        CASE "Tor2_program".program.numerKroku OF
	            7243, 7320:
	                "Cip".obiekt[#nr].procedura := 3;
	            ELSE
	                "Cip".obiekt[#nr].procedura := 0;
	        END_CASE;
	        
	    CASE "Cip".obiekt[#nr].procedura OF
	    2:
	    //set - warunki dla wejścia funkcji Set
	    "Cip".obiekt[#nr].SetReset.czasDoSet := 10;
	    "Cip".obiekt[#nr].SetReset.inSet :=
	    "Cip".obiekt["Cip".tor[0].zbiorniczekDozowaniaKwasu.czujnikDolnegoPoziomu].hmiPotwWysterowania = 1
	    AND ("Tor2_RecepturyStacjaMycia".numerKrokuMycia = 4);
	    
	    //reset - warunki dla wejścia funkcji Reset
	    "Cip".obiekt[#nr].SetReset.czasDoReset := 0;
	    "Cip".obiekt[#nr].SetReset.inReset :=
	    "Cip".obiekt["Cip".tor[0].zbiorniczekDozowaniaKwasu.czujnikDolnegoPoziomu].hmiPotwWysterowania = 0
	    OR ("Tor2_RecepturyStacjaMycia".numerKrokuMycia = 3);
	    
	    //załaczanie
	    "Cip".obiekt[#nr].Flipaj.czas_ON := 300;
	    "Cip".obiekt[#nr].Flipaj.czas_OFF := 100;
	    "Cip".obiekt[#nr].Flipaj.ile_petli := 999;
	    "Cip".obiekt[#nr].Flipaj.in := "Cip".obiekt[#nr].SetReset.wyjście;
	    "Cip".obiekt[#nr].inStartAuto := "Cip".obiekt[#nr].Flipaj.Q;
	    
	    //wysterowanie
	    "Cip".obiekt[#nr].inZadaneWysterowanieAuto := 100.0;
	    
	    3:
	    //set - warunki dla wejścia funkcji Set
	    "Cip".obiekt[#nr].SetReset.czasDoSet := 100;
	    "Cip".obiekt[#nr].SetReset.inSet :=
	    "Cip".obiekt["Cip".tor[0].zbiorniczekDozowaniaKwasu.czujnikDolnegoPoziomu].hmiPotwWysterowania = 1
	    AND ("Tor2_RecepturyStacjaMycia".numerKrokuMycia = 4) //warunki dla toru Cip1
	    AND ("Cip".obiekt["Cip".tor[2].przewodnośćNaPowrocie].WartośćPomiaru <
	    "Tor2_RecepturyStacjaMycia".Receptura[#aktualnyNumerReceptury].Krok[#aktualnyKrokMycia].PM[11]);
	    
	    
	    //reset - warunki dla wejścia funkcji Reset
	    "Cip".obiekt[#nr].SetReset.czasDoReset := 0;
	    "Cip".obiekt[#nr].SetReset.inReset :=
	    "Cip".obiekt["Cip".tor[0].zbiorniczekDozowaniaKwasu.czujnikDolnegoPoziomu].hmiPotwWysterowania = 0
	    OR ("Tor2_RecepturyStacjaMycia".numerKrokuMycia = 3) //warunki dla toru Cip1
	    OR ("Cip".obiekt["Cip".tor[2].przewodnośćNaPowrocie].WartośćPomiaru >=
	    "Tor2_RecepturyStacjaMycia".Receptura[#aktualnyNumerReceptury].Krok[#aktualnyKrokMycia].PM[11]);
	    
	    //załaczanie
	    "Cip".obiekt[#nr].Flipaj.czas_ON := REAL_TO_INT(
	                                                    "Tor2_RecepturyStacjaMycia".
	                                                    Receptura[#aktualnyNumerReceptury].
	                                                    Krok[#aktualnyKrokMycia].PM[26] * 10);
	    "Cip".obiekt[#nr].Flipaj.czas_OFF := REAL_TO_INT(
	                                                     "Tor2_RecepturyStacjaMycia".
	                                                     Receptura[#aktualnyNumerReceptury].
	                                                     Krok[#aktualnyKrokMycia].PM[27] * 10);
	    "Cip".obiekt[#nr].Flipaj.ile_petli :=
	    REAL_TO_INT("Tor2_RecepturyStacjaMycia".Receptura[#aktualnyNumerReceptury].Krok[#aktualnyKrokMycia].PM[20] /
	                ("Tor2_RecepturyStacjaMycia".Receptura[#aktualnyNumerReceptury].Krok[#aktualnyKrokMycia].PM[26] +
	                "Tor2_RecepturyStacjaMycia".Receptura[#aktualnyNumerReceptury].Krok[#aktualnyKrokMycia].PM[27] + 1.0));
	    "Cip".obiekt[#nr].Flipaj.in := "Cip".obiekt[#nr].SetReset.wyjście;
	    "Cip".obiekt[#nr].inStartAuto := "Cip".obiekt[#nr].Flipaj.Q;
	    
	    //wysterowanie
	    "Cip".obiekt[#nr].inZadaneWysterowanieAuto := 100.0;
	0:
	    "Cip".obiekt[#nr].Flipaj.in := 0;
	 
	    END_CASE;
	    
	    END_REGION
	    
	    REGION POMPKA DOZOWANIA DEZYNFEKANTU W LINIE
	    
	        #nr := "Cip".tor[2].pompkaDozowaniaDezynfekantuwLinię;
	        
	        CASE "Tor2_program".program.numerKroku OF
	            7281:
	                "Cip".obiekt[#nr].procedura := 2;
	            ELSE
	                "Cip".obiekt[#nr].procedura := 0;
	        END_CASE;
	        
	    CASE "Cip".obiekt[#nr].procedura OF
	    2:
	    
	    //
	    //załaczanie
	    "Cip".obiekt[#nr].Flipaj.czas_ON := REAL_TO_INT(
	                                                  "Tor2_RecepturyStacjaMycia".
	                                                  Receptura[#aktualnyNumerReceptury].
	                                                  Krok[#aktualnyKrokMycia].PM[26] * 10);
	    "Cip".obiekt[#nr].Flipaj.czas_OFF := REAL_TO_INT(
	                                                   "Tor2_RecepturyStacjaMycia".
	                                                   Receptura[#aktualnyNumerReceptury].
	                                                   Krok[#aktualnyKrokMycia].PM[27] * 10);
	  "Cip".obiekt[#nr].Flipaj.ile_petli := 999;
	    // REAL_TO_INT("Tor2_RecepturyStacjaMycia".Receptura[#aktualnyNumerReceptury].Krok[#aktualnyKrokMycia].PM[20] /
	    //             ("Tor2_RecepturyStacjaMycia".Receptura[#aktualnyNumerReceptury].Krok[#aktualnyKrokMycia].PM[26] +
	    //             "Tor2_RecepturyStacjaMycia".Receptura[#aktualnyNumerReceptury].Krok[#aktualnyKrokMycia].PM[27] + 1.0));
	    
	    ;
	    "Cip".obiekt[#nr].Flipaj.in := 1;
	    "Cip".obiekt[#nr].inStartAuto := "Cip".obiekt[#nr].Flipaj.Q;
	
	    0:
	    "Cip".obiekt[#nr].Flipaj.in := 0;
	    END_CASE;
	END_REGION
	REGION zawor  DOZOWANIA DEZYNFEKANTU W LINIE
	    
	    #nr := "Cip".tor[2].zawórDozowaniaDezynfekantuwLinię;
	    
	    CASE "Tor2_program".program.numerKroku OF
	        7281:
	            "Cip".obiekt[#nr].procedura := 2;
	        ELSE
	            "Cip".obiekt[#nr].procedura := 0;
	    END_CASE;
	    
	    CASE "Cip".obiekt[#nr].procedura OF
	        2:
	            
	            //
	            //załaczanie
	      
	            
	            ;
	           
